	UF : 0, UT : 6,		CONFIG : 'N U T, 0, 0, 0',
	X =  -103.237  mm,	Y =   -367.062  mm,	Z =   -236.482  mm,
	W =  90.000 deg,	P =   0.000 deg,	R =   90.000 deg
};
P[2666]{
   GP1:
	UF : 0, UT : 6,		CONFIG : 'N U T, 0, 0, 0',
	X =  -103.796  mm,	Y =   -367.200  mm,	Z =   -236.035  mm,
	W =  90.000 deg,	P =   0.000 deg,	R =   90.000 deg
};
P[2667]{
   GP1:
	UF : 0, UT : 6,		CONFIG : 'N U T, 0, 0, 0',
	X =  -109.111  mm,	Y =   -370.387  mm,	Z =   -236.321  mm,
	W =  90.000 deg,	P =   0.000 deg,	R =   90.000 deg
};
P[2668]{
   GP1:
	UF : 0, UT : 6,		CONFIG : 'N U T, 0, 0, 0',
	X =  -109.874  mm,	Y =   -370.891  mm,	Z =   -236.475  mm,
	W =  90.000 deg,	P =   0.000 deg,	R =   90.000 deg
};
P[2669]{
   GP1:
	UF : 0, UT : 6,		CONFIG : 'N U T, 0, 0, 0',
	X =  -111.510  mm,	Y =   -371.847  mm,	Z =   -236.505  mm,
	W =  90.000 deg,	P =   0.000 deg,	R =   90.000 deg
};
P[2670]{
   GP1:
	UF : 0, UT : 6,		CONFIG : 'N U T, 0, 0, 0',
	X =  -113.758  mm,	Y =   -372.951  mm,	Z =   -236.032  mm,
	W =  90.000 deg,	P =   0.000 deg,	R =   90.000 deg
};
P[2671]{
   GP1:
	UF : 0, UT : 6,		CONFIG : 'N U T, 0, 0, 0',
	X =  -115.678  mm,	Y =   -374.223  mm,	Z =   -236.429  mm,
	W =  90.000 deg,	P =   0.000 deg,	R =   90.000 deg
};
P[2672]{
   GP1:
	UF : 0, UT : 6,		CONFIG : 'N U T, 0, 0, 0',
	X =  -117.192  mm,	Y =   -375.019  mm,	Z =   -236.240  mm,
	W =  90.000 deg,	P =   0.000 deg,	R =   90.000 deg
};
P[2673]{
   GP1:
	UF : 0, UT : 6,		CONFIG : 'N U T, 0, 0, 0',
	X =  -118.313  mm,	Y =   -375.755  mm,	Z =   -236.454  mm,
	W =  90.000 deg,	P =   0.000 deg,	R =   90.000 deg
};
P[2674]{
   GP1:
	UF : 0, UT : 6,		CONFIG : 'N U T, 0, 0, 0',
	X =  -120.295  mm,	Y =   -376.722  mm,	Z =   -236.025  mm,
	W =  90.000 deg,	P =   0.000 deg,	R =   90.000 deg
};
P[2675]{
   GP1:
	UF : 0, UT : 6,		CONFIG : 'N U T, 0, 0, 0',
	X =  -121.428  mm,	Y =   -377.386  mm,	Z =   -236.049  mm,
	W =  90.000 deg,	P =   0.000 deg,	R =   90.000 deg
};
P[2676]{
   GP1:
	UF : 0, UT : 6,		CONFIG : 'N U T, 0, 0, 0',
	X =  -123.033  mm,	Y =   -378.483  mm,	Z =   -236.461  mm,
	W =  90.000 deg,	P =   0.000 deg,	R =   90.000 deg
};
P[2677]{
   GP1:
	UF : 0, UT : 6,		CONFIG : 'N U T, 0, 0, 0',
	X =  -123.863  mm,	Y =   -378.861  mm,	Z =   -236.217  mm,
	W =  90.000 deg,	P =   0.000 deg,	R =   90.000 deg
};
P[2678]{
   GP1:
	UF : 0, UT : 6,		CONFIG : 'N U T, 0, 0, 0',
	X =  -125.601  mm,	Y =   -379.960  mm,	Z =   -236.448  mm,
	W =  90.000 deg,	P =   0.000 deg,	R =   90.000 deg
};
P[2679]{
   GP1:
	UF : 0, UT : 6,		CONFIG : 'N U T, 0, 0, 0',
	X =  -128.227  mm,	Y =   -381.434  mm,	Z =   -236.345  mm,
	W =  90.000 deg,	P =   0.000 deg,	R =   90.000 deg
};
P[2680]{
   GP1:
	UF : 0, UT : 6,		CONFIG : 'N U T, 0, 0, 0',
	X =  -131.933  mm,	Y =   -383.507  mm,	Z =   -236.183  mm,
	W =  90.000 deg,	P =   0.000 deg,	R =   90.000 deg
};
P[2681]{
   GP1:
	UF : 0, UT : 6,		CONFIG : 'N U T, 0, 0, 0',
	X =  -134.089  mm,	Y =   -385.044  mm,	Z =   -236.339  mm,
	W =  90.000 deg,	P =   0.000 deg,	R =   90.000 deg
};
P[2682]{
   GP1:
	UF : 0, UT : 6,		CONFIG : 'N U T, 0, 0, 0',
	X =  -136.292  mm,	Y =   -387.219  mm,	Z =   -236.419  mm,
	W =  90.000 deg,	P =   0.000 deg,	R =   90.000 deg
};
P[2683]{
   GP1:
	UF : 0, UT : 6,		CONFIG : 'N U T, 0, 0, 0',
	X =  -137.707  mm,	Y =   -389.283  mm,	Z =   -236.379  mm,
	W =  90.000 deg,	P =   0.000 deg,	R =   90.000 deg
};
P[2684]{
   GP1:
	UF : 0, UT : 6,		CONFIG : 'N U T, 0, 0, 0',
	X =  -138.543  mm,	Y =   -391.394  mm,	Z =   -236.512  mm,
	W =  90.000 deg,	P =   0.000 deg,	R =   90.000 deg
};
P[2685]{
   GP1:
	UF : 0, UT : 6,		CONFIG : 'N U T, 0, 0, 0',
	X =  -138.974  mm,	Y =   -392.288  mm,	Z =   -236.247  mm,
	W =  90.000 deg,	P =   0.000 deg,	R =   90.000 deg
};
P[2686]{
   GP1:
	UF : 0, UT : 6,		CONFIG : 'N U T, 0, 0, 0',
	X =  -139.171  mm,	Y =   -393.080  mm,	Z =   -236.154  mm,
	W =  90.000 deg,	P =   0.000 deg,	R =   90.000 deg
};
P[2687]{
   GP1:
	UF : 0, UT : 6,		CONFIG : 'N U T, 0, 0, 0',
	X =  -139.217  mm,	Y =   -394.462  mm,	Z =   -236.503  mm,
	W =  90.000 deg,	P =   0.000 deg,	R =   90.000 deg
};
P[2688]{
   GP1:
	UF : 0, UT : 6,		CONFIG : 'N U T, 0, 0, 0',
	X =  -139.347  mm,	Y =   -395.646  mm,	Z =   -236.277  mm,
	W =  90.000 deg,	P =   0.000 deg,	R =   90.000 deg
};
P[2689]{
   GP1:
	UF : 0, UT : 6,		CONFIG : 'N U T, 0, 0, 0',
	X =  -139.228  mm,	Y =   -396.334  mm,	Z =   -236.466  mm,
	W =  90.000 deg,	P =   0.000 deg,	R =   90.000 deg
};
P[2690]{
   GP1:
	UF : 0, UT : 6,		CONFIG : 'N U T, 0, 0, 0',
	X =  -139.026  mm,	Y =   -398.050  mm,	Z =   -236.504  mm,
	W =  90.000 deg,	P =   0.000 deg,	R =   90.000 deg
};
P[2691]{
   GP1:
	UF : 0, UT : 6,		CONFIG : 'N U T, 0, 0, 0',
	X =  -138.894  mm,	Y =   -399.249  mm,	Z =   -236.149  mm,
	W =  90.000 deg,	P =   0.000 deg,	R =   90.000 deg
};
P[2692]{
   GP1:
	UF : 0, UT : 6,		CONFIG : 'N U T, 0, 0, 0',
	X =  -138.534  mm,	Y =   -400.086  mm,	Z =   -236.490  mm,
	W =  90.000 deg,	P =   0.000 deg,	R =   90.000 deg
};
P[2693]{
   GP1:
	UF : 0, UT : 6,		CONFIG : 'N U T, 0, 0, 0',
	X =  -138.293  mm,	Y =   -400.993  mm,	Z =   -236.111  mm,
	W =  90.000 deg,	P =   0.000 deg,	R =   90.000 deg
};
P[2694]{
   GP1:
	UF : 0, UT : 6,		CONFIG : 'N U T, 0, 0, 0',
	X =  -132.435  mm,	Y =   -411.328  mm,	Z =   -236.323  mm,
	W =  90.000 deg,	P =   0.000 deg,	R =   90.000 deg
};
P[2695]{
   GP1:
	UF : 0, UT : 6,		CONFIG : 'N U T, 0, 0, 0',
	X =  -131.602  mm,	Y =   -412.647  mm,	Z =   -236.497  mm,
	W =  90.000 deg,	P =   0.000 deg,	R =   90.000 deg
};
P[2696]{
   GP1:
	UF : 0, UT : 6,		CONFIG : 'N U T, 0, 0, 0',
	X =  -131.076  mm,	Y =   -413.576  mm,	Z =   -236.473  mm,
	W =  90.000 deg,	P =   0.000 deg,	R =   90.000 deg
};
P[2697]{
   GP1:
	UF : 0, UT : 6,		CONFIG : 'N U T, 0, 0, 0',
	X =  -130.720  mm,	Y =   -414.277  mm,	Z =   -236.355  mm,
	W =  90.000 deg,	P =   0.000 deg,	R =   90.000 deg
};
P[2698]{
   GP1:
	UF : 0, UT : 6,		CONFIG : 'N U T, 0, 0, 0',
	X =  -129.684  mm,	Y =   -415.969  mm,	Z =   -236.496  mm,
	W =  90.000 deg,	P =   0.000 deg,	R =   90.000 deg
};
P[2699]{
   GP1:
	UF : 0, UT : 6,		CONFIG : 'N U T, 0, 0, 0',
	X =  -128.664  mm,	Y =   -417.827  mm,	Z =   -236.369  mm,
	W =  90.000 deg,	P =   0.000 deg,	R =   90.000 deg
};
P[2700]{
   GP1:
	UF : 0, UT : 6,		CONFIG : 'N U T, 0, 0, 0',
	X =  -127.347  mm,	Y =   -420.040  mm,	Z =   -236.463  mm,
	W =  90.000 deg,	P =   0.000 deg,	R =   90.000 deg
};
P[2701]{
   GP1:
	UF : 0, UT : 6,		CONFIG : 'N U T, 0, 0, 0',
	X =  -126.510  mm,	Y =   -421.475  mm,	Z =   -236.485  mm,
	W =  90.000 deg,	P =   0.000 deg,	R =   90.000 deg
};
P[2702]{
   GP1:
	UF : 0, UT : 6,		CONFIG : 'N U T, 0, 0, 0',
	X =  -125.653  mm,	Y =   -423.090  mm,	Z =   -236.300  mm,
	W =  90.000 deg,	P =   0.000 deg,	R =   90.000 deg
};
P[2703]{
   GP1:
	UF : 0, UT : 6,		CONFIG : 'N U T, 0, 0, 0',
	X =  -124.246  mm,	Y =   -425.539  mm,	Z =   -236.286  mm,
	W =  90.000 deg,	P =   0.000 deg,	R =   90.000 deg
};
P[2704]{
   GP1:
	UF : 0, UT : 6,		CONFIG : 'N U T, 0, 0, 0',
	X =  -122.328  mm,	Y =   -428.699  mm,	Z =   -236.513  mm,
	W =  90.000 deg,	P =   0.000 deg,	R =   90.000 deg
};
P[2705]{
   GP1:
	UF : 0, UT : 6,		CONFIG : 'N U T, 0, 0, 0',
	X =  -121.006  mm,	Y =   -431.158  mm,	Z =   -236.273  mm,
	W =  90.000 deg,	P =   0.000 deg,	R =   90.000 deg
};
P[2706]{
   GP1:
	UF : 0, UT : 6,		CONFIG : 'N U T, 0, 0, 0',
	X =  -117.398  mm,	Y =   -437.502  mm,	Z =   -236.140  mm,
	W =  90.000 deg,	P =   0.000 deg,	R =   90.000 deg
};
P[2707]{
   GP1:
	UF : 0, UT : 6,		CONFIG : 'N U T, 0, 0, 0',
	X =  -116.351  mm,	Y =   -439.270  mm,	Z =   -236.205  mm,
	W =  90.000 deg,	P =   0.000 deg,	R =   90.000 deg
};
P[2708]{
   GP1:
	UF : 0, UT : 6,		CONFIG : 'N U T, 0, 0, 0',
	X =  -115.892  mm,	Y =   -439.878  mm,	Z =   -236.465  mm,
	W =  90.000 deg,	P =   0.000 deg,	R =   90.000 deg
};
P[2709]{
   GP1:
	UF : 0, UT : 6,		CONFIG : 'N U T, 0, 0, 0',
	X =  -112.701  mm,	Y =   -445.426  mm,	Z =   -236.435  mm,
	W =  90.000 deg,	P =   0.000 deg,	R =   90.000 deg
};
P[2710]{
   GP1:
	UF : 0, UT : 6,		CONFIG : 'N U T, 0, 0, 0',
	X =  -111.296  mm,	Y =   -448.012  mm,	Z =   -236.222  mm,
	W =  90.000 deg,	P =   0.000 deg,	R =   90.000 deg
};
P[2711]{
   GP1:
	UF : 0, UT : 6,		CONFIG : 'N U T, 0, 0, 0',
	X =  -110.621  mm,	Y =   -448.979  mm,	Z =   -236.505  mm,
	W =  90.000 deg,	P =   0.000 deg,	R =   90.000 deg
};
P[2712]{
   GP1:
	UF : 0, UT : 6,		CONFIG : 'N U T, 0, 0, 0',
	X =  -109.896  mm,	Y =   -450.279  mm,	Z =   -236.445  mm,
	W =  90.000 deg,	P =   0.000 deg,	R =   90.000 deg
};
P[2713]{
   GP1:
	UF : 0, UT : 6,		CONFIG : 'N U T, 0, 0, 0',
	X =  -109.523  mm,	Y =   -451.116  mm,	Z =   -236.175  mm,
	W =  90.000 deg,	P =   0.000 deg,	R =   90.000 deg
};
P[2714]{
   GP1:
	UF : 0, UT : 6,		CONFIG : 'N U T, 0, 0, 0',
	X =  -109.072  mm,	Y =   -451.738  mm,	Z =   -236.398  mm,
	W =  90.000 deg,	P =   0.000 deg,	R =   90.000 deg
};
P[2715]{
   GP1:
	UF : 0, UT : 6,		CONFIG : 'N U T, 0, 0, 0',
	X =  -108.224  mm,	Y =   -453.286  mm,	Z =   -236.287  mm,
	W =  90.000 deg,	P =   0.000 deg,	R =   90.000 deg
};
P[2716]{
   GP1:
	UF : 0, UT : 6,		CONFIG : 'N U T, 0, 0, 0',
	X =  -107.392  mm,	Y =   -454.819  mm,	Z =   -236.157  mm,
	W =  90.000 deg,	P =   0.000 deg,	R =   90.000 deg
};
P[2717]{
   GP1:
	UF : 0, UT : 6,		CONFIG : 'N U T, 0, 0, 0',
	X =  -104.616  mm,	Y =   -459.487  mm,	Z =   -236.353  mm,
	W =  90.000 deg,	P =   0.000 deg,	R =   90.000 deg
};
P[2718]{
   GP1:
	UF : 0, UT : 6,		CONFIG : 'N U T, 0, 0, 0',
	X =  -103.935  mm,	Y =   -460.905  mm,	Z =   -236.019  mm,
	W =  90.000 deg,	P =   0.000 deg,	R =   90.000 deg
};
P[2719]{
   GP1:
	UF : 0, UT : 6,		CONFIG : 'N U T, 0, 0, 0',
	X =  -103.296  mm,	Y =   -461.877  mm,	Z =   -236.210  mm,
	W =  90.000 deg,	P =   0.000 deg,	R =   90.000 deg
};
P[2720]{
   GP1:
	UF : 0, UT : 6,		CONFIG : 'N U T, 0, 0, 0',
	X =  -102.498  mm,	Y =   -463.081  mm,	Z =   -236.458  mm,
	W =  90.000 deg,	P =   0.000 deg,	R =   90.000 deg
};
P[2721]{
   GP1:
	UF : 0, UT : 6,		CONFIG : 'N U T, 0, 0, 0',
	X =  -102.062  mm,	Y =   -463.796  mm,	Z =   -236.514  mm,
	W =  90.000 deg,	P =   0.000 deg,	R =   90.000 deg
};
P[2722]{
   GP1:
	UF : 0, UT : 6,		CONFIG : 'N U T, 0, 0, 0',
	X =  -98.860  mm,	Y =   -469.387  mm,	Z =   -236.452  mm,
	W =  90.000 deg,	P =   0.000 deg,	R =   90.000 deg
};
P[2723]{
   GP1:
	UF : 0, UT : 6,		CONFIG : 'N U T, 0, 0, 0',
	X =  -97.430  mm,	Y =   -472.003  mm,	Z =   -236.256  mm,
	W =  90.000 deg,	P =   0.000 deg,	R =   90.000 deg
};
P[2724]{
   GP1:
	UF : 0, UT : 6,		CONFIG : 'N U T, 0, 0, 0',
	X =  -95.657  mm,	Y =   -474.990  mm,	Z =   -236.371  mm,
	W =  90.000 deg,	P =   0.000 deg,	R =   90.000 deg
};
P[2725]{
   GP1:
	UF : 0, UT : 6,		CONFIG : 'N U T, 0, 0, 0',
	X =  -95.143  mm,	Y =   -475.820  mm,	Z =   -236.456  mm,
	W =  90.000 deg,	P =   0.000 deg,	R =   90.000 deg
};
P[2726]{
   GP1:
	UF : 0, UT : 6,		CONFIG : 'N U T, 0, 0, 0',
	X =  -94.054  mm,	Y =   -477.851  mm,	Z =   -236.254  mm,
	W =  90.000 deg,	P =   0.000 deg,	R =   90.000 deg
};
P[2727]{
   GP1:
	UF : 0, UT : 6,		CONFIG : 'N U T, 0, 0, 0',
	X =  -92.555  mm,	Y =   -480.264  mm,	Z =   -236.509  mm,
	W =  90.000 deg,	P =   0.000 deg,	R =   90.000 deg
};
P[2728]{
   GP1:
	UF : 0, UT : 6,		CONFIG : 'N U T, 0, 0, 0',
	X =  -90.494  mm,	Y =   -484.012  mm,	Z =   -236.260  mm,
	W =  90.000 deg,	P =   0.000 deg,	R =   90.000 deg
};
P[2729]{
   GP1:
	UF : 0, UT : 6,		CONFIG : 'N U T, 0, 0, 0',
	X =  -89.771  mm,	Y =   -485.179  mm,	Z =   -236.380  mm,
	W =  90.000 deg,	P =   0.000 deg,	R =   90.000 deg
};
P[2730]{
   GP1:
	UF : 0, UT : 6,		CONFIG : 'N U T, 0, 0, 0',
	X =  -88.079  mm,	Y =   -488.059  mm,	Z =   -236.451  mm,
	W =  90.000 deg,	P =   0.000 deg,	R =   90.000 deg
};
P[2731]{
   GP1:
	UF : 0, UT : 6,		CONFIG : 'N U T, 0, 0, 0',
	X =  -83.696  mm,	Y =   -495.609  mm,	Z =   -236.506  mm,
	W =  90.000 deg,	P =   0.000 deg,	R =   90.000 deg
};
P[2732]{
   GP1:
	UF : 0, UT : 6,		CONFIG : 'N U T, 0, 0, 0',
	X =  -83.326  mm,	Y =   -496.356  mm,	Z =   -236.359  mm,
	W =  90.000 deg,	P =   0.000 deg,	R =   90.000 deg
};
P[2733]{
   GP1:
	UF : 0, UT : 6,		CONFIG : 'N U T, 0, 0, 0',
	X =  -82.778  mm,	Y =   -497.396  mm,	Z =   -236.232  mm,
	W =  90.000 deg,	P =   0.000 deg,	R =   90.000 deg
};
P[2734]{
   GP1:
	UF : 0, UT : 6,		CONFIG : 'N U T, 0, 0, 0',
	X =  -82.192  mm,	Y =   -498.250  mm,	Z =   -236.458  mm,
	W =  90.000 deg,	P =   0.000 deg,	R =   90.000 deg
};
P[2735]{
   GP1:
	UF : 0, UT : 6,		CONFIG : 'N U T, 0, 0, 0',
	X =  -79.146  mm,	Y =   -503.762  mm,	Z =   -236.125  mm,
	W =  90.000 deg,	P =   0.000 deg,	R =   90.000 deg
};
P[2736]{
   GP1:
	UF : 0, UT : 6,		CONFIG : 'N U T, 0, 0, 0',
	X =  -77.301  mm,	Y =   -506.708  mm,	Z =   -236.474  mm,
	W =  90.000 deg,	P =   0.000 deg,	R =   90.000 deg
};
P[2737]{
   GP1:
	UF : 0, UT : 6,		CONFIG : 'N U T, 0, 0, 0',
	X =  -75.967  mm,	Y =   -509.301  mm,	Z =   -236.079  mm,
	W =  90.000 deg,	P =   0.000 deg,	R =   90.000 deg
};
P[2738]{
   GP1:
	UF : 0, UT : 6,		CONFIG : 'N U T, 0, 0, 0',
	X =  -74.945  mm,	Y =   -510.996  mm,	Z =   -236.183  mm,
	W =  90.000 deg,	P =   0.000 deg,	R =   90.000 deg
};
P[2739]{
   GP1:
	UF : 0, UT : 6,		CONFIG : 'N U T, 0, 0, 0',
	X =  -71.961  mm,	Y =   -516.089  mm,	Z =   -236.291  mm,
	W =  90.000 deg,	P =   0.000 deg,	R =   90.000 deg
};
P[2740]{
   GP1:
	UF : 0, UT : 6,		CONFIG : 'N U T, 0, 0, 0',
	X =  -70.926  mm,	Y =   -517.733  mm,	Z =   -236.499  mm,
	W =  90.000 deg,	P =   0.000 deg,	R =   90.000 deg
};
P[2741]{
   GP1:
	UF : 0, UT : 6,		CONFIG : 'N U T, 0, 0, 0',
	X =  -70.119  mm,	Y =   -519.466  mm,	Z =   -236.027  mm,
	W =  90.000 deg,	P =   0.000 deg,	R =   90.000 deg
};
P[2742]{
   GP1:
	UF : 0, UT : 6,		CONFIG : 'N U T, 0, 0, 0',
	X =  -67.807  mm,	Y =   -523.183  mm,	Z =   -236.430  mm,
	W =  90.000 deg,	P =   0.000 deg,	R =   90.000 deg
};
P[2743]{
   GP1:
	UF : 0, UT : 6,		CONFIG : 'N U T, 0, 0, 0',
	X =  -67.049  mm,	Y =   -524.711  mm,	Z =   -236.128  mm,
	W =  90.000 deg,	P =   0.000 deg,	R =   90.000 deg
};
P[2744]{
   GP1:
	UF : 0, UT : 6,		CONFIG : 'N U T, 0, 0, 0',
	X =  -63.701  mm,	Y =   -530.270  mm,	Z =   -236.462  mm,
	W =  90.000 deg,	P =   0.000 deg,	R =   90.000 deg
};
P[2745]{
   GP1:
	UF : 0, UT : 6,		CONFIG : 'N U T, 0, 0, 0',
	X =  -63.119  mm,	Y =   -531.321  mm,	Z =   -236.403  mm,
	W =  90.000 deg,	P =   0.000 deg,	R =   90.000 deg
};
P[2746]{
   GP1:
	UF : 0, UT : 6,		CONFIG : 'N U T, 0, 0, 0',
	X =  -61.469  mm,	Y =   -534.194  mm,	Z =   -236.385  mm,
	W =  90.000 deg,	P =   0.000 deg,	R =   90.000 deg
};
P[2747]{
   GP1:
	UF : 0, UT : 6,		CONFIG : 'N U T, 0, 0, 0',
	X =  -61.266  mm,	Y =   -534.788  mm,	Z =   -236.042  mm,
	W =  90.000 deg,	P =   0.000 deg,	R =   90.000 deg
};
P[2748]{
   GP1:
	UF : 0, UT : 6,		CONFIG : 'N U T, 0, 0, 0',
	X =  -60.082  mm,	Y =   -536.624  mm,	Z =   -236.345  mm,
	W =  90.000 deg,	P =   0.000 deg,	R =   90.000 deg
};
P[2749]{
   GP1:
	UF : 0, UT : 6,		CONFIG : 'N U T, 0, 0, 0',
	X =  -59.497  mm,	Y =   -537.677  mm,	Z =   -236.288  mm,
	W =  90.000 deg,	P =   0.000 deg,	R =   90.000 deg
};
P[2750]{
   GP1:
	UF : 0, UT : 6,		CONFIG : 'N U T, 0, 0, 0',
	X =  -59.054  mm,	Y =   -538.435  mm,	Z =   -236.301  mm,
	W =  90.000 deg,	P =   0.000 deg,	R =   90.000 deg
};
P[2751]{
   GP1:
	UF : 0, UT : 6,		CONFIG : 'N U T, 0, 0, 0',
	X =  -56.974  mm,	Y =   -542.109  mm,	Z =   -236.201  mm,
	W =  90.000 deg,	P =   0.000 deg,	R =   90.000 deg
};
P[2752]{
   GP1:
	UF : 0, UT : 6,		CONFIG : 'N U T, 0, 0, 0',
	X =  -56.447  mm,	Y =   -542.963  mm,	Z =   -236.281  mm,
	W =  90.000 deg,	P =   0.000 deg,	R =   90.000 deg
};
P[2753]{
   GP1:
	UF : 0, UT : 6,		CONFIG : 'N U T, 0, 0, 0',
	X =  -55.849  mm,	Y =   -543.939  mm,	Z =   -236.367  mm,
	W =  90.000 deg,	P =   0.000 deg,	R =   90.000 deg
};
P[2754]{
   GP1:
	UF : 0, UT : 6,		CONFIG : 'N U T, 0, 0, 0',
	X =  -54.722  mm,	Y =   -545.925  mm,	Z =   -236.316  mm,
	W =  90.000 deg,	P =   0.000 deg,	R =   90.000 deg
};
P[2755]{
   GP1:
	UF : 0, UT : 6,		CONFIG : 'N U T, 0, 0, 0',
	X =  -53.820  mm,	Y =   -547.403  mm,	Z =   -236.437  mm,
	W =  90.000 deg,	P =   0.000 deg,	R =   90.000 deg
};
P[2756]{
   GP1:
	UF : 0, UT : 6,		CONFIG : 'N U T, 0, 0, 0',
	X =  -51.903  mm,	Y =   -550.957  mm,	Z =   -236.109  mm,
	W =  90.000 deg,	P =   0.000 deg,	R =   90.000 deg
};
P[2757]{
   GP1:
	UF : 0, UT : 6,		CONFIG : 'N U T, 0, 0, 0',
	X =  -50.467  mm,	Y =   -553.413  mm,	Z =   -236.152  mm,
	W =  90.000 deg,	P =   0.000 deg,	R =   90.000 deg
};
P[2758]{
   GP1:
	UF : 0, UT : 6,		CONFIG : 'N U T, 0, 0, 0',
	X =  -49.404  mm,	Y =   -555.025  mm,	Z =   -236.475  mm,
	W =  90.000 deg,	P =   0.000 deg,	R =   90.000 deg
};
P[2759]{
   GP1:
	UF : 0, UT : 6,		CONFIG : 'N U T, 0, 0, 0',
	X =  -47.513  mm,	Y =   -558.279  mm,	Z =   -236.503  mm,
	W =  90.000 deg,	P =   0.000 deg,	R =   90.000 deg
};
P[2760]{
   GP1:
	UF : 0, UT : 6,		CONFIG : 'N U T, 0, 0, 0',
	X =  -47.011  mm,	Y =   -559.184  mm,	Z =   -236.452  mm,
	W =  90.000 deg,	P =   0.000 deg,	R =   90.000 deg
};
P[2761]{
   GP1:
	UF : 0, UT : 6,		CONFIG : 'N U T, 0, 0, 0',
	X =  -45.707  mm,	Y =   -561.524  mm,	Z =   -236.340  mm,
	W =  90.000 deg,	P =   0.000 deg,	R =   90.000 deg
};
P[2762]{
   GP1:
	UF : 0, UT : 6,		CONFIG : 'N U T, 0, 0, 0',
	X =  -44.786  mm,	Y =   -563.328  mm,	Z =   -236.045  mm,
	W =  90.000 deg,	P =   0.000 deg,	R =   90.000 deg
};
P[2763]{
   GP1:
	UF : 0, UT : 6,		CONFIG : 'N U T, 0, 0, 0',
	X =  -43.612  mm,	Y =   -565.119  mm,	Z =   -236.386  mm,
	W =  90.000 deg,	P =   0.000 deg,	R =   90.000 deg
};
P[2764]{
   GP1:
	UF : 0, UT : 6,		CONFIG : 'N U T, 0, 0, 0',
	X =  -43.076  mm,	Y =   -565.989  mm,	Z =   -236.466  mm,
	W =  90.000 deg,	P =   0.000 deg,	R =   90.000 deg
};
P[2765]{
   GP1:
	UF : 0, UT : 6,		CONFIG : 'N U T, 0, 0, 0',
	X =  -40.936  mm,	Y =   -569.844  mm,	Z =   -236.260  mm,
	W =  90.000 deg,	P =   0.000 deg,	R =   90.000 deg
};
P[2766]{
   GP1:
	UF : 0, UT : 6,		CONFIG : 'N U T, 0, 0, 0',
	X =  -40.504  mm,	Y =   -570.459  mm,	Z =   -236.446  mm,
	W =  90.000 deg,	P =   0.000 deg,	R =   90.000 deg
};
P[2767]{
   GP1:
	UF : 0, UT : 6,		CONFIG : 'N U T, 0, 0, 0',
	X =  -39.086  mm,	Y =   -572.957  mm,	Z =   -236.386  mm,
	W =  90.000 deg,	P =   0.000 deg,	R =   90.000 deg
};
P[2768]{
   GP1:
	UF : 0, UT : 6,		CONFIG : 'N U T, 0, 0, 0',
	X =  -36.165  mm,	Y =   -577.983  mm,	Z =   -236.433  mm,
	W =  90.000 deg,	P =   0.000 deg,	R =   90.000 deg
};
P[2769]{
   GP1:
	UF : 0, UT : 6,		CONFIG : 'N U T, 0, 0, 0',
	X =  -35.589  mm,	Y =   -578.926  mm,	Z =   -236.508  mm,
	W =  90.000 deg,	P =   0.000 deg,	R =   90.000 deg
};
P[2770]{
   GP1:
	UF : 0, UT : 6,		CONFIG : 'N U T, 0, 0, 0',
	X =  -30.957  mm,	Y =   -587.282  mm,	Z =   -236.040  mm,
	W =  90.000 deg,	P =   0.000 deg,	R =   90.000 deg
};
P[2771]{
   GP1:
	UF : 0, UT : 6,		CONFIG : 'N U T, 0, 0, 0',
	X =  -29.354  mm,	Y =   -589.787  mm,	Z =   -236.423  mm,
	W =  90.000 deg,	P =   0.000 deg,	R =   90.000 deg
};
P[2772]{
   GP1:
	UF : 0, UT : 6,		CONFIG : 'N U T, 0, 0, 0',
	X =  -26.877  mm,	Y =   -594.032  mm,	Z =   -236.483  mm,
	W =  90.000 deg,	P =   0.000 deg,	R =   90.000 deg
};
P[2773]{
   GP1:
	UF : 0, UT : 6,		CONFIG : 'N U T, 0, 0, 0',
	X =  -23.884  mm,	Y =   -599.221  mm,	Z =   -236.478  mm,
	W =  90.000 deg,	P =   0.000 deg,	R =   90.000 deg
};
P[2774]{
   GP1:
	UF : 0, UT : 6,		CONFIG : 'N U T, 0, 0, 0',
	X =  -22.979  mm,	Y =   -600.863  mm,	Z =   -236.375  mm,
	W =  90.000 deg,	P =   0.000 deg,	R =   90.000 deg
};
P[2775]{
   GP1:
	UF : 0, UT : 6,		CONFIG : 'N U T, 0, 0, 0',
	X =  -22.245  mm,	Y =   -602.071  mm,	Z =   -236.459  mm,
	W =  90.000 deg,	P =   0.000 deg,	R =   90.000 deg
};
P[2776]{
   GP1:
	UF : 0, UT : 6,		CONFIG : 'N U T, 0, 0, 0',
	X =  -21.779  mm,	Y =   -602.853  mm,	Z =   -236.496  mm,
	W =  90.000 deg,	P =   0.000 deg,	R =   90.000 deg
};
P[2777]{
   GP1:
	UF : 0, UT : 6,		CONFIG : 'N U T, 0, 0, 0',
	X =  -20.072  mm,	Y =   -605.860  mm,	Z =   -236.425  mm,
	W =  90.000 deg,	P =   0.000 deg,	R =   90.000 deg
};
P[2778]{
   GP1:
	UF : 0, UT : 6,		CONFIG : 'N U T, 0, 0, 0',
	X =  -17.813  mm,	Y =   -609.858  mm,	Z =   -236.308  mm,
	W =  90.000 deg,	P =   0.000 deg,	R =   90.000 deg
};
P[2779]{
   GP1:
	UF : 0, UT : 6,		CONFIG : 'N U T, 0, 0, 0',
	X =  -16.783  mm,	Y =   -611.767  mm,	Z =   -236.131  mm,
	W =  90.000 deg,	P =   0.000 deg,	R =   90.000 deg
};
P[2780]{
   GP1:
	UF : 0, UT : 6,		CONFIG : 'N U T, 0, 0, 0',
	X =  -16.133  mm,	Y =   -612.837  mm,	Z =   -236.208  mm,
	W =  90.000 deg,	P =   0.000 deg,	R =   90.000 deg
};
P[2781]{
   GP1:
	UF : 0, UT : 6,		CONFIG : 'N U T, 0, 0, 0',
	X =  -15.576  mm,	Y =   -613.717  mm,	Z =   -236.326  mm,
	W =  90.000 deg,	P =   0.000 deg,	R =   90.000 deg
};
P[2782]{
   GP1:
	UF : 0, UT : 6,		CONFIG : 'N U T, 0, 0, 0',
	X =  -13.580  mm,	Y =   -617.138  mm,	Z =   -236.378  mm,
	W =  90.000 deg,	P =   0.000 deg,	R =   90.000 deg
};
P[2783]{
   GP1:
	UF : 0, UT : 6,		CONFIG : 'N U T, 0, 0, 0',
	X =  -12.725  mm,	Y =   -618.540  mm,	Z =   -236.487  mm,
	W =  90.000 deg,	P =   0.000 deg,	R =   90.000 deg
};
P[2784]{
   GP1:
	UF : 0, UT : 6,		CONFIG : 'N U T, 0, 0, 0',
	X =  -12.420  mm,	Y =   -619.263  mm,	Z =   -236.216  mm,
	W =  90.000 deg,	P =   0.000 deg,	R =   90.000 deg
};
P[2785]{
   GP1:
	UF : 0, UT : 6,		CONFIG : 'N U T, 0, 0, 0',
	X =  -11.625  mm,	Y =   -620.474  mm,	Z =   -236.448  mm,
	W =  90.000 deg,	P =   0.000 deg,	R =   90.000 deg
};
P[2786]{
   GP1:
	UF : 0, UT : 6,		CONFIG : 'N U T, 0, 0, 0',
	X =  -8.389  mm,	Y =   -626.060  mm,	Z =   -236.474  mm,
	W =  90.000 deg,	P =   0.000 deg,	R =   90.000 deg
};
P[2787]{
   GP1:
	UF : 0, UT : 6,		CONFIG : 'N U T, 0, 0, 0',
	X =  -6.891  mm,	Y =   -628.784  mm,	Z =   -236.289  mm,
	W =  90.000 deg,	P =   0.000 deg,	R =   90.000 deg
};
P[2788]{
   GP1:
	UF : 0, UT : 6,		CONFIG : 'N U T, 0, 0, 0',
	X =  -6.304  mm,	Y =   -629.768  mm,	Z =   -236.336  mm,
	W =  90.000 deg,	P =   0.000 deg,	R =   90.000 deg
};
P[2789]{
   GP1:
	UF : 0, UT : 6,		CONFIG : 'N U T, 0, 0, 0',
	X =  -5.756  mm,	Y =   -630.621  mm,	Z =   -236.473  mm,
	W =  90.000 deg,	P =   0.000 deg,	R =   90.000 deg
};
P[2790]{
   GP1:
	UF : 0, UT : 6,		CONFIG : 'N U T, 0, 0, 0',
	X =  -3.081  mm,	Y =   -635.232  mm,	Z =   -236.502  mm,
	W =  90.000 deg,	P =   0.000 deg,	R =   90.000 deg
};
P[2791]{
   GP1:
	UF : 0, UT : 6,		CONFIG : 'N U T, 0, 0, 0',
	X =  -2.279  mm,	Y =   -636.663  mm,	Z =   -236.443  mm,
	W =  90.000 deg,	P =   0.000 deg,	R =   90.000 deg
};
P[2792]{
   GP1:
	UF : 0, UT : 6,		CONFIG : 'N U T, 0, 0, 0',
	X =  -0.761  mm,	Y =   -639.336  mm,	Z =   -236.383  mm,
	W =  90.000 deg,	P =   0.000 deg,	R =   90.000 deg
};
P[2793]{
   GP1:
	UF : 0, UT : 6,		CONFIG : 'N U T, 0, 0, 0',
	X =  0.858  mm,	Y =   -642.148  mm,	Z =   -236.369  mm,
	W =  90.000 deg,	P =   0.000 deg,	R =   90.000 deg
};
P[2794]{
   GP1:
	UF : 0, UT : 6,		CONFIG : 'N U T, 0, 0, 0',
	X =  1.759  mm,	Y =   -643.769  mm,	Z =   -236.287  mm,
	W =  90.000 deg,	P =   0.000 deg,	R =   90.000 deg
};
P[2795]{
   GP1:
	UF : 0, UT : 6,		CONFIG : 'N U T, 0, 0, 0',
	X =  3.576  mm,	Y =   -646.947  mm,	Z =   -236.243  mm,
	W =  90.000 deg,	P =   0.000 deg,	R =   90.000 deg
};
P[2796]{
   GP1:
	UF : 0, UT : 6,		CONFIG : 'N U T, 0, 0, 0',
	X =  4.161  mm,	Y =   -647.944  mm,	Z =   -236.266  mm,
	W =  90.000 deg,	P =   0.000 deg,	R =   90.000 deg
};
P[2797]{
   GP1:
	UF : 0, UT : 6,		CONFIG : 'N U T, 0, 0, 0',
	X =  4.658  mm,	Y =   -648.779  mm,	Z =   -236.302  mm,
	W =  90.000 deg,	P =   0.000 deg,	R =   90.000 deg
};
P[2798]{
   GP1:
	UF : 0, UT : 6,		CONFIG : 'N U T, 0, 0, 0',
	X =  5.200  mm,	Y =   -649.689  mm,	Z =   -236.343  mm,
	W =  90.000 deg,	P =   0.000 deg,	R =   90.000 deg
};
P[2799]{
   GP1:
	UF : 0, UT : 6,		CONFIG : 'N U T, 0, 0, 0',
	X =  5.838  mm,	Y =   -650.769  mm,	Z =   -236.379  mm,
	W =  90.000 deg,	P =   0.000 deg,	R =   90.000 deg
};
P[2800]{
   GP1:
	UF : 0, UT : 6,		CONFIG : 'N U T, 0, 0, 0',
	X =  9.409  mm,	Y =   -656.940  mm,	Z =   -236.398  mm,
	W =  90.000 deg,	P =   0.000 deg,	R =   90.000 deg
};
P[2801]{
   GP1:
	UF : 0, UT : 6,		CONFIG : 'N U T, 0, 0, 0',
	X =  11.270  mm,	Y =   -660.160  mm,	Z =   -236.402  mm,
	W =  90.000 deg,	P =   0.000 deg,	R =   90.000 deg
};
P[2802]{
   GP1:
	UF : 0, UT : 6,		CONFIG : 'N U T, 0, 0, 0',
	X =  12.634  mm,	Y =   -662.517  mm,	Z =   -236.408  mm,
	W =  90.000 deg,	P =   0.000 deg,	R =   90.000 deg
};
P[2803]{
   GP1:
	UF : 0, UT : 6,		CONFIG : 'N U T, 0, 0, 0',
	X =  13.698  mm,	Y =   -664.325  mm,	Z =   -236.457  mm,
	W =  90.000 deg,	P =   0.000 deg,	R =   90.000 deg
};
P[2804]{
   GP1:
	UF : 0, UT : 6,		CONFIG : 'N U T, 0, 0, 0',
	X =  14.024  mm,	Y =   -665.020  mm,	Z =   -236.275  mm,
	W =  90.000 deg,	P =   0.000 deg,	R =   90.000 deg
};
P[2805]{
   GP1:
	UF : 0, UT : 6,		CONFIG : 'N U T, 0, 0, 0',
	X =  15.603  mm,	Y =   -667.779  mm,	Z =   -236.241  mm,
	W =  90.000 deg,	P =   0.000 deg,	R =   90.000 deg
};
P[2806]{
   GP1:
	UF : 0, UT : 6,		CONFIG : 'N U T, 0, 0, 0',
	X =  16.111  mm,	Y =   -668.721  mm,	Z =   -236.153  mm,
	W =  90.000 deg,	P =   0.000 deg,	R =   90.000 deg
};
P[2807]{
   GP1:
	UF : 0, UT : 6,		CONFIG : 'N U T, 0, 0, 0',
	X =  16.623  mm,	Y =   -669.667  mm,	Z =   -236.072  mm,
	W =  90.000 deg,	P =   0.000 deg,	R =   90.000 deg
};
P[2808]{
   GP1:
	UF : 0, UT : 6,		CONFIG : 'N U T, 0, 0, 0',
	X =  18.028  mm,	Y =   -672.101  mm,	Z =   -236.068  mm,
	W =  90.000 deg,	P =   0.000 deg,	R =   90.000 deg
};
P[2809]{
   GP1:
	UF : 0, UT : 6,		CONFIG : 'N U T, 0, 0, 0',
	X =  18.530  mm,	Y =   -672.742  mm,	Z =   -236.391  mm,
	W =  90.000 deg,	P =   0.000 deg,	R =   90.000 deg
};
P[2810]{
   GP1:
	UF : 0, UT : 6,		CONFIG : 'N U T, 0, 0, 0',
	X =  20.590  mm,	Y =   -676.325  mm,	Z =   -236.365  mm,
	W =  90.000 deg,	P =   0.000 deg,	R =   90.000 deg
};
P[2811]{
   GP1:
	UF : 0, UT : 6,		CONFIG : 'N U T, 0, 0, 0',
	X =  22.083  mm,	Y =   -679.038  mm,	Z =   -236.189  mm,
	W =  90.000 deg,	P =   0.000 deg,	R =   90.000 deg
};
P[2812]{
   GP1:
	UF : 0, UT : 6,		CONFIG : 'N U T, 0, 0, 0',
	X =  23.478  mm,	Y =   -681.252  mm,	Z =   -236.473  mm,
	W =  90.000 deg,	P =   0.000 deg,	R =   90.000 deg
};
P[2813]{
   GP1:
	UF : 0, UT : 6,		CONFIG : 'N U T, 0, 0, 0',
	X =  24.055  mm,	Y =   -682.577  mm,	Z =   -236.016  mm,
	W =  90.000 deg,	P =   0.000 deg,	R =   90.000 deg
};
P[2814]{
   GP1:
	UF : 0, UT : 6,		CONFIG : 'N U T, 0, 0, 0',
	X =  27.203  mm,	Y =   -687.875  mm,	Z =   -236.234  mm,
	W =  90.000 deg,	P =   0.000 deg,	R =   90.000 deg
};
P[2815]{
   GP1:
	UF : 0, UT : 6,		CONFIG : 'N U T, 0, 0, 0',
	X =  27.873  mm,	Y =   -688.847  mm,	Z =   -236.496  mm,
	W =  90.000 deg,	P =   0.000 deg,	R =   90.000 deg
};
P[2816]{
   GP1:
	UF : 0, UT : 6,		CONFIG : 'N U T, 0, 0, 0',
	X =  28.459  mm,	Y =   -689.879  mm,	Z =   -236.471  mm,
	W =  90.000 deg,	P =   0.000 deg,	R =   90.000 deg
};
P[2817]{
   GP1:
	UF : 0, UT : 6,		CONFIG : 'N U T, 0, 0, 0',
	X =  29.323  mm,	Y =   -691.489  mm,	Z =   -236.312  mm,
	W =  90.000 deg,	P =   0.000 deg,	R =   90.000 deg
};
P[2818]{
   GP1:
	UF : 0, UT : 6,		CONFIG : 'N U T, 0, 0, 0',
	X =  30.796  mm,	Y =   -694.114  mm,	Z =   -236.209  mm,
	W =  90.000 deg,	P =   0.000 deg,	R =   90.000 deg
};
P[2819]{
   GP1:
	UF : 0, UT : 6,		CONFIG : 'N U T, 0, 0, 0',
	X =  32.101  mm,	Y =   -696.258  mm,	Z =   -236.372  mm,
	W =  90.000 deg,	P =   0.000 deg,	R =   90.000 deg
};
P[2820]{
   GP1:
	UF : 0, UT : 6,		CONFIG : 'N U T, 0, 0, 0',
	X =  34.273  mm,	Y =   -699.958  mm,	Z =   -236.458  mm,
	W =  90.000 deg,	P =   0.000 deg,	R =   90.000 deg
};
P[2821]{
   GP1:
	UF : 0, UT : 6,		CONFIG : 'N U T, 0, 0, 0',
	X =  35.034  mm,	Y =   -701.310  mm,	Z =   -236.409  mm,
	W =  90.000 deg,	P =   0.000 deg,	R =   90.000 deg
};
P[2822]{
   GP1:
	UF : 0, UT : 6,		CONFIG : 'N U T, 0, 0, 0',
	X =  35.645  mm,	Y =   -702.304  mm,	Z =   -236.268  mm,
	W =  90.000 deg,	P =   0.000 deg,	R =   90.000 deg
};
P[2823]{
   GP1:
	UF : 0, UT : 6,		CONFIG : 'N U T, 0, 0, 0',
	X =  36.316  mm,	Y =   -703.207  mm,	Z =   -236.328  mm,
	W =  90.000 deg,	P =   0.000 deg,	R =   90.000 deg
};
P[2824]{
   GP1:
	UF : 0, UT : 6,		CONFIG : 'N U T, 0, 0, 0',
	X =  37.230  mm,	Y =   -704.410  mm,	Z =   -236.133  mm,
	W =  90.000 deg,	P =   0.000 deg,	R =   90.000 deg
};
P[2825]{
   GP1:
	UF : 0, UT : 6,		CONFIG : 'N U T, 0, 0, 0',
	X =  38.416  mm,	Y =   -705.323  mm,	Z =   -236.491  mm,
	W =  90.000 deg,	P =   0.000 deg,	R =   90.000 deg
};
P[2826]{
   GP1:
	UF : 0, UT : 6,		CONFIG : 'N U T, 0, 0, 0',
	X =  39.372  mm,	Y =   -706.033  mm,	Z =   -236.512  mm,
	W =  90.000 deg,	P =   0.000 deg,	R =   90.000 deg
};
P[2827]{
   GP1:
	UF : 0, UT : 6,		CONFIG : 'N U T, 0, 0, 0',
	X =  40.316  mm,	Y =   -706.802  mm,	Z =   -236.215  mm,
	W =  90.000 deg,	P =   0.000 deg,	R =   90.000 deg
};
P[2828]{
   GP1:
	UF : 0, UT : 6,		CONFIG : 'N U T, 0, 0, 0',
	X =  45.468  mm,	Y =   -708.560  mm,	Z =   -236.089  mm,
	W =  90.000 deg,	P =   0.000 deg,	R =   90.000 deg
};
P[2829]{
   GP1:
	UF : 0, UT : 6,		CONFIG : 'N U T, 0, 0, 0',
	X =  46.166  mm,	Y =   -708.584  mm,	Z =   -236.188  mm,
	W =  90.000 deg,	P =   0.000 deg,	R =   90.000 deg
};
P[2830]{
   GP1:
	UF : 0, UT : 6,		CONFIG : 'N U T, 0, 0, 0',
	X =  47.620  mm,	Y =   -708.412  mm,	Z =   -236.473  mm,
	W =  90.000 deg,	P =   0.000 deg,	R =   90.000 deg
};
P[2831]{
   GP1:
	UF : 0, UT : 6,		CONFIG : 'N U T, 0, 0, 0',
	X =  48.514  mm,	Y =   -708.561  mm,	Z =   -236.085  mm,
	W =  90.000 deg,	P =   0.000 deg,	R =   90.000 deg
};
P[2832]{
   GP1:
	UF : 0, UT : 6,		CONFIG : 'N U T, 0, 0, 0',
	X =  49.691  mm,	Y =   -708.218  mm,	Z =   -236.321  mm,
	W =  90.000 deg,	P =   0.000 deg,	R =   90.000 deg
};
P[2833]{
   GP1:
	UF : 0, UT : 6,		CONFIG : 'N U T, 0, 0, 0',
	X =  52.176  mm,	Y =   -707.394  mm,	Z =   -236.458  mm,
	W =  90.000 deg,	P =   0.000 deg,	R =   90.000 deg
};
P[2834]{
   GP1:
	UF : 0, UT : 6,		CONFIG : 'N U T, 0, 0, 0',
	X =  56.284  mm,	Y =   -705.282  mm,	Z =   -236.360  mm,
	W =  90.000 deg,	P =   0.000 deg,	R =   90.000 deg
};
P[2835]{
   GP1:
	UF : 0, UT : 6,		CONFIG : 'N U T, 0, 0, 0',
	X =  59.075  mm,	Y =   -703.766  mm,	Z =   -236.129  mm,
	W =  90.000 deg,	P =   0.000 deg,	R =   90.000 deg
};
P[2836]{
   GP1:
	UF : 0, UT : 6,		CONFIG : 'N U T, 0, 0, 0',
	X =  59.898  mm,	Y =   -703.189  mm,	Z =   -236.376  mm,
	W =  90.000 deg,	P =   0.000 deg,	R =   90.000 deg
};
P[2837]{
   GP1:
	UF : 0, UT : 6,		CONFIG : 'N U T, 0, 0, 0',
	X =  61.634  mm,	Y =   -702.160  mm,	Z =   -236.438  mm,
	W =  90.000 deg,	P =   0.000 deg,	R =   90.000 deg
};
P[2838]{
   GP1:
	UF : 0, UT : 6,		CONFIG : 'N U T, 0, 0, 0',
	X =  63.182  mm,	Y =   -701.329  mm,	Z =   -236.288  mm,
	W =  90.000 deg,	P =   0.000 deg,	R =   90.000 deg
};
P[2839]{
   GP1:
	UF : 0, UT : 6,		CONFIG : 'N U T, 0, 0, 0',
	X =  66.400  mm,	Y =   -699.411  mm,	Z =   -236.431  mm,
	W =  90.000 deg,	P =   0.000 deg,	R =   90.000 deg
};
P[2840]{
   GP1:
	UF : 0, UT : 6,		CONFIG : 'N U T, 0, 0, 0',
	X =  68.844  mm,	Y =   -698.171  mm,	Z =   -236.017  mm,
	W =  90.000 deg,	P =   0.000 deg,	R =   90.000 deg
};
P[2841]{
   GP1:
	UF : 0, UT : 6,		CONFIG : 'N U T, 0, 0, 0',
	X =  69.752  mm,	Y =   -697.447  mm,	Z =   -236.500  mm,
	W =  90.000 deg,	P =   0.000 deg,	R =   90.000 deg
};
P[2842]{
   GP1:
	UF : 0, UT : 6,		CONFIG : 'N U T, 0, 0, 0',
	X =  71.033  mm,	Y =   -696.871  mm,	Z =   -236.105  mm,
	W =  90.000 deg,	P =   0.000 deg,	R =   90.000 deg
};
P[2843]{
   GP1:
	UF : 0, UT : 6,		CONFIG : 'N U T, 0, 0, 0',
	X =  79.303  mm,	Y =   -692.067  mm,	Z =   -236.174  mm,
	W =  90.000 deg,	P =   0.000 deg,	R =   90.000 deg
};
P[2844]{
   GP1:
	UF : 0, UT : 6,		CONFIG : 'N U T, 0, 0, 0',
	X =  80.219  mm,	Y =   -691.581  mm,	Z =   -236.072  mm,
	W =  90.000 deg,	P =   0.000 deg,	R =   90.000 deg
};
P[2845]{
   GP1:
	UF : 0, UT : 6,		CONFIG : 'N U T, 0, 0, 0',
	X =  82.107  mm,	Y =   -690.492  mm,	Z =   -236.067  mm,
	W =  90.000 deg,	P =   0.000 deg,	R =   90.000 deg
};
P[2846]{
   GP1:
	UF : 0, UT : 6,		CONFIG : 'N U T, 0, 0, 0',
	X =  82.790  mm,	Y =   -689.951  mm,	Z =   -236.423  mm,
	W =  90.000 deg,	P =   0.000 deg,	R =   90.000 deg
};
P[2847]{
   GP1:
	UF : 0, UT : 6,		CONFIG : 'N U T, 0, 0, 0',
	X =  84.311  mm,	Y =   -689.078  mm,	Z =   -236.410  mm,
	W =  90.000 deg,	P =   0.000 deg,	R =   90.000 deg
};
P[2848]{
   GP1:
	UF : 0, UT : 6,		CONFIG : 'N U T, 0, 0, 0',
	X =  87.841  mm,	Y =   -687.160  mm,	Z =   -236.120  mm,
	W =  90.000 deg,	P =   0.000 deg,	R =   90.000 deg
};
P[2849]{
   GP1:
	UF : 0, UT : 6,		CONFIG : 'N U T, 0, 0, 0',
	X =  90.417  mm,	Y =   -685.662  mm,	Z =   -236.144  mm,
	W =  90.000 deg,	P =   0.000 deg,	R =   90.000 deg
};
P[2850]{
   GP1:
	UF : 0, UT : 6,		CONFIG : 'N U T, 0, 0, 0',
	X =  92.018  mm,	Y =   -684.683  mm,	Z =   -236.277  mm,
	W =  90.000 deg,	P =   0.000 deg,	R =   90.000 deg
};
P[2851]{
   GP1:
	UF : 0, UT : 6,		CONFIG : 'N U T, 0, 0, 0',
	X =  95.149  mm,	Y =   -682.789  mm,	Z =   -236.487  mm,
	W =  90.000 deg,	P =   0.000 deg,	R =   90.000 deg
};
P[2852]{
   GP1:
	UF : 0, UT : 6,		CONFIG : 'N U T, 0, 0, 0',
	X =  96.225  mm,	Y =   -682.338  mm,	Z =   -236.074  mm,
	W =  90.000 deg,	P =   0.000 deg,	R =   90.000 deg
};
P[2853]{
   GP1:
	UF : 0, UT : 6,		CONFIG : 'N U T, 0, 0, 0',
	X =  97.254  mm,	Y =   -681.639  mm,	Z =   -236.329  mm,
	W =  90.000 deg,	P =   0.000 deg,	R =   90.000 deg
};
P[2854]{
   GP1:
	UF : 0, UT : 6,		CONFIG : 'N U T, 0, 0, 0',
	X =  97.958  mm,	Y =   -681.341  mm,	Z =   -236.066  mm,
	W =  90.000 deg,	P =   0.000 deg,	R =   90.000 deg
};
P[2855]{
   GP1:
	UF : 0, UT : 6,		CONFIG : 'N U T, 0, 0, 0',
	X =  109.694  mm,	Y =   -674.564  mm,	Z =   -236.067  mm,
	W =  90.000 deg,	P =   0.000 deg,	R =   90.000 deg
};
P[2856]{
   GP1:
	UF : 0, UT : 6,		CONFIG : 'N U T, 0, 0, 0',
	X =  114.432  mm,	Y =   -671.794  mm,	Z =   -236.150  mm,
	W =  90.000 deg,	P =   0.000 deg,	R =   90.000 deg
};
P[2857]{
   GP1:
	UF : 0, UT : 6,		CONFIG : 'N U T, 0, 0, 0',
	X =  118.155  mm,	Y =   -669.576  mm,	Z =   -236.314  mm,
	W =  90.000 deg,	P =   0.000 deg,	R =   90.000 deg
};
P[2858]{
   GP1:
	UF : 0, UT : 6,		CONFIG : 'N U T, 0, 0, 0',
	X =  119.202  mm,	Y =   -668.923  mm,	Z =   -236.432  mm,
	W =  90.000 deg,	P =   0.000 deg,	R =   90.000 deg
};
P[2859]{
   GP1:
	UF : 0, UT : 6,		CONFIG : 'N U T, 0, 0, 0',
	X =  124.199  mm,	Y =   -666.158  mm,	Z =   -236.141  mm,
	W =  90.000 deg,	P =   0.000 deg,	R =   90.000 deg
};
P[2860]{
   GP1:
	UF : 0, UT : 6,		CONFIG : 'N U T, 0, 0, 0',
	X =  128.547  mm,	Y =   -663.511  mm,	Z =   -236.473  mm,
	W =  90.000 deg,	P =   0.000 deg,	R =   90.000 deg
};
P[2861]{
   GP1:
	UF : 0, UT : 6,		CONFIG : 'N U T, 0, 0, 0',
	X =  130.385  mm,	Y =   -662.451  mm,	Z =   -236.470  mm,
	W =  90.000 deg,	P =   0.000 deg,	R =   90.000 deg
};
P[2862]{
   GP1:
	UF : 0, UT : 6,		CONFIG : 'N U T, 0, 0, 0',
	X =  131.198  mm,	Y =   -662.021  mm,	Z =   -236.374  mm,
	W =  90.000 deg,	P =   0.000 deg,	R =   90.000 deg
};
P[2863]{
   GP1:
	UF : 0, UT : 6,		CONFIG : 'N U T, 0, 0, 0',
	X =  133.444  mm,	Y =   -660.671  mm,	Z =   -236.505  mm,
	W =  90.000 deg,	P =   0.000 deg,	R =   90.000 deg
};
P[2864]{
   GP1:
	UF : 0, UT : 6,		CONFIG : 'N U T, 0, 0, 0',
	X =  136.895  mm,	Y =   -658.782  mm,	Z =   -236.252  mm,
	W =  90.000 deg,	P =   0.000 deg,	R =   90.000 deg
};
P[2865]{
   GP1:
	UF : 0, UT : 6,		CONFIG : 'N U T, 0, 0, 0',
	X =  139.530  mm,	Y =   -657.201  mm,	Z =   -236.398  mm,
	W =  90.000 deg,	P =   0.000 deg,	R =   90.000 deg
};
P[2866]{
   GP1:
	UF : 0, UT : 6,		CONFIG : 'N U T, 0, 0, 0',
	X =  140.472  mm,	Y =   -656.701  mm,	Z =   -236.291  mm,
	W =  90.000 deg,	P =   0.000 deg,	R =   90.000 deg
};
P[2867]{
   GP1:
	UF : 0, UT : 6,		CONFIG : 'N U T, 0, 0, 0',
	X =  142.309  mm,	Y =   -655.675  mm,	Z =   -236.206  mm,
	W =  90.000 deg,	P =   0.000 deg,	R =   90.000 deg
};
P[2868]{
   GP1:
	UF : 0, UT : 6,		CONFIG : 'N U T, 0, 0, 0',
	X =  144.452  mm,	Y =   -654.460  mm,	Z =   -236.153  mm,
	W =  90.000 deg,	P =   0.000 deg,	R =   90.000 deg
};
P[2869]{
   GP1:
	UF : 0, UT : 6,		CONFIG : 'N U T, 0, 0, 0',
	X =  145.368  mm,	Y =   -653.865  mm,	Z =   -236.312  mm,
	W =  90.000 deg,	P =   0.000 deg,	R =   90.000 deg
};
P[2870]{
   GP1:
	UF : 0, UT : 6,		CONFIG : 'N U T, 0, 0, 0',
	X =  148.587  mm,	Y =   -652.078  mm,	Z =   -236.139  mm,
	W =  90.000 deg,	P =   0.000 deg,	R =   90.000 deg
};
P[2871]{
   GP1:
	UF : 0, UT : 6,		CONFIG : 'N U T, 0, 0, 0',
	X =  150.438  mm,	Y =   -650.983  mm,	Z =   -236.201  mm,
	W =  90.000 deg,	P =   0.000 deg,	R =   90.000 deg
};
P[2872]{
   GP1:
	UF : 0, UT : 6,		CONFIG : 'N U T, 0, 0, 0',
	X =  152.235  mm,	Y =   -649.851  mm,	Z =   -236.430  mm,
	W =  90.000 deg,	P =   0.000 deg,	R =   90.000 deg
};
P[2873]{
   GP1:
	UF : 0, UT : 6,		CONFIG : 'N U T, 0, 0, 0',
	X =  154.556  mm,	Y =   -648.513  mm,	Z =   -236.428  mm,
	W =  90.000 deg,	P =   0.000 deg,	R =   90.000 deg
};
P[2874]{
   GP1:
	UF : 0, UT : 6,		CONFIG : 'N U T, 0, 0, 0',
	X =  155.199  mm,	Y =   -648.213  mm,	Z =   -236.255  mm,
	W =  90.000 deg,	P =   0.000 deg,	R =   90.000 deg
};
P[2875]{
   GP1:
	UF : 0, UT : 6,		CONFIG : 'N U T, 0, 0, 0',
	X =  157.457  mm,	Y =   -646.981  mm,	Z =   -236.079  mm,
	W =  90.000 deg,	P =   0.000 deg,	R =   90.000 deg
};
P[2876]{
   GP1:
	UF : 0, UT : 6,		CONFIG : 'N U T, 0, 0, 0',
	X =  159.587  mm,	Y =   -645.594  mm,	Z =   -236.459  mm,
	W =  90.000 deg,	P =   0.000 deg,	R =   90.000 deg
};
P[2877]{
   GP1:
	UF : 0, UT : 6,		CONFIG : 'N U T, 0, 0, 0',
	X =  160.338  mm,	Y =   -645.329  mm,	Z =   -236.051  mm,
	W =  90.000 deg,	P =   0.000 deg,	R =   90.000 deg
};
P[2878]{
   GP1:
	UF : 0, UT : 6,		CONFIG : 'N U T, 0, 0, 0',
	X =  163.247  mm,	Y =   -643.545  mm,	Z =   -236.305  mm,
	W =  90.000 deg,	P =   0.000 deg,	R =   90.000 deg
};
P[2879]{
   GP1:
	UF : 0, UT : 6,		CONFIG : 'N U T, 0, 0, 0',
	X =  163.919  mm,	Y =   -643.248  mm,	Z =   -236.085  mm,
	W =  90.000 deg,	P =   0.000 deg,	R =   90.000 deg
};
P[2880]{
   GP1:
	UF : 0, UT : 6,		CONFIG : 'N U T, 0, 0, 0',
	X =  165.705  mm,	Y =   -642.087  mm,	Z =   -236.398  mm,
	W =  90.000 deg,	P =   0.000 deg,	R =   90.000 deg
};
P[2881]{
   GP1:
	UF : 0, UT : 6,		CONFIG : 'N U T, 0, 0, 0',
	X =  167.372  mm,	Y =   -641.217  mm,	Z =   -236.176  mm,
	W =  90.000 deg,	P =   0.000 deg,	R =   90.000 deg
};
P[2882]{
   GP1:
	UF : 0, UT : 6,		CONFIG : 'N U T, 0, 0, 0',
	X =  168.552  mm,	Y =   -640.521  mm,	Z =   -236.212  mm,
	W =  90.000 deg,	P =   0.000 deg,	R =   90.000 deg
};
P[2883]{
   GP1:
	UF : 0, UT : 6,		CONFIG : 'N U T, 0, 0, 0',
	X =  169.884  mm,	Y =   -639.665  mm,	Z =   -236.422  mm,
	W =  90.000 deg,	P =   0.000 deg,	R =   90.000 deg
};
P[2884]{
   GP1:
	UF : 0, UT : 6,		CONFIG : 'N U T, 0, 0, 0',
	X =  171.046  mm,	Y =   -639.027  mm,	Z =   -236.340  mm,
	W =  90.000 deg,	P =   0.000 deg,	R =   90.000 deg
};
P[2885]{
   GP1:
	UF : 0, UT : 6,		CONFIG : 'N U T, 0, 0, 0',
	X =  173.896  mm,	Y =   -637.386  mm,	Z =   -236.330  mm,
	W =  90.000 deg,	P =   0.000 deg,	R =   90.000 deg
};
P[2886]{
   GP1:
	UF : 0, UT : 6,		CONFIG : 'N U T, 0, 0, 0',
	X =  175.734  mm,	Y =   -636.399  mm,	Z =   -236.152  mm,
	W =  90.000 deg,	P =   0.000 deg,	R =   90.000 deg
};
P[2887]{
   GP1:
	UF : 0, UT : 6,		CONFIG : 'N U T, 0, 0, 0',
	X =  178.103  mm,	Y =   -634.901  mm,	Z =   -236.465  mm,
	W =  90.000 deg,	P =   0.000 deg,	R =   90.000 deg
};
P[2888]{
   GP1:
	UF : 0, UT : 6,		CONFIG : 'N U T, 0, 0, 0',
	X =  179.069  mm,	Y =   -634.471  mm,	Z =   -236.155  mm,
	W =  90.000 deg,	P =   0.000 deg,	R =   90.000 deg
};
P[2889]{
   GP1:
	UF : 0, UT : 6,		CONFIG : 'N U T, 0, 0, 0',
	X =  180.259  mm,	Y =   -633.839  mm,	Z =   -236.021  mm,
	W =  90.000 deg,	P =   0.000 deg,	R =   90.000 deg
};
P[2890]{
   GP1:
	UF : 0, UT : 6,		CONFIG : 'N U T, 0, 0, 0',
	X =  181.350  mm,	Y =   -633.209  mm,	Z =   -236.022  mm,
	W =  90.000 deg,	P =   0.000 deg,	R =   90.000 deg
};
P[2891]{
   GP1:
	UF : 0, UT : 6,		CONFIG : 'N U T, 0, 0, 0',
	X =  188.115  mm,	Y =   -629.190  mm,	Z =   -236.296  mm,
	W =  90.000 deg,	P =   0.000 deg,	R =   90.000 deg
};
P[2892]{
   GP1:
	UF : 0, UT : 6,		CONFIG : 'N U T, 0, 0, 0',
	X =  194.718  mm,	Y =   -625.303  mm,	Z =   -236.477  mm,
	W =  90.000 deg,	P =   0.000 deg,	R =   90.000 deg
};
P[2893]{
   GP1:
	UF : 0, UT : 6,		CONFIG : 'N U T, 0, 0, 0',
	X =  195.641  mm,	Y =   -624.763  mm,	Z =   -236.494  mm,
	W =  90.000 deg,	P =   0.000 deg,	R =   90.000 deg
};
P[2894]{
   GP1:
	UF : 0, UT : 6,		CONFIG : 'N U T, 0, 0, 0',
	X =  196.542  mm,	Y =   -624.285  mm,	Z =   -236.391  mm,
	W =  90.000 deg,	P =   0.000 deg,	R =   90.000 deg
};
P[2895]{
   GP1:
	UF : 0, UT : 6,		CONFIG : 'N U T, 0, 0, 0',
	X =  198.006  mm,	Y =   -623.439  mm,	Z =   -236.393  mm,
	W =  90.000 deg,	P =   0.000 deg,	R =   90.000 deg
};
P[2896]{
   GP1:
	UF : 0, UT : 6,		CONFIG : 'N U T, 0, 0, 0',
	X =  198.990  mm,	Y =   -622.855  mm,	Z =   -236.432  mm,
	W =  90.000 deg,	P =   0.000 deg,	R =   90.000 deg
};
P[2897]{
   GP1:
	UF : 0, UT : 6,		CONFIG : 'N U T, 0, 0, 0',
	X =  201.991  mm,	Y =   -621.238  mm,	Z =   -236.150  mm,
	W =  90.000 deg,	P =   0.000 deg,	R =   90.000 deg
};
P[2898]{
   GP1:
	UF : 0, UT : 6,		CONFIG : 'N U T, 0, 0, 0',
	X =  203.362  mm,	Y =   -620.476  mm,	Z =   -236.080  mm,
	W =  90.000 deg,	P =   0.000 deg,	R =   90.000 deg
};
P[2899]{
   GP1:
	UF : 0, UT : 6,		CONFIG : 'N U T, 0, 0, 0',
	X =  205.942  mm,	Y =   -618.867  mm,	Z =   -236.366  mm,
	W =  90.000 deg,	P =   0.000 deg,	R =   90.000 deg
};
P[2900]{
   GP1:
	UF : 0, UT : 6,		CONFIG : 'N U T, 0, 0, 0',
	X =  206.618  mm,	Y =   -618.506  mm,	Z =   -236.298  mm,
	W =  90.000 deg,	P =   0.000 deg,	R =   90.000 deg
};
P[2901]{
   GP1:
	UF : 0, UT : 6,		CONFIG : 'N U T, 0, 0, 0',
	X =  208.093  mm,	Y =   -617.590  mm,	Z =   -236.453  mm,
	W =  90.000 deg,	P =   0.000 deg,	R =   90.000 deg
};
P[2902]{
   GP1:
	UF : 0, UT : 6,		CONFIG : 'N U T, 0, 0, 0',
	X =  209.850  mm,	Y =   -616.555  mm,	Z =   -236.502  mm,
	W =  90.000 deg,	P =   0.000 deg,	R =   90.000 deg
};
P[2903]{
   GP1:
	UF : 0, UT : 6,		CONFIG : 'N U T, 0, 0, 0',
	X =  211.605  mm,	Y =   -615.684  mm,	Z =   -236.157  mm,
	W =  90.000 deg,	P =   0.000 deg,	R =   90.000 deg
};
P[2904]{
   GP1:
	UF : 0, UT : 6,		CONFIG : 'N U T, 0, 0, 0',
	X =  212.954  mm,	Y =   -614.933  mm,	Z =   -236.090  mm,
	W =  90.000 deg,	P =   0.000 deg,	R =   90.000 deg
};
P[2905]{
   GP1:
	UF : 0, UT : 6,		CONFIG : 'N U T, 0, 0, 0',
	X =  214.059  mm,	Y =   -614.147  mm,	Z =   -236.449  mm,
	W =  90.000 deg,	P =   0.000 deg,	R =   90.000 deg
};
P[2906]{
   GP1:
	UF : 0, UT : 6,		CONFIG : 'N U T, 0, 0, 0',
	X =  216.542  mm,	Y =   -612.809  mm,	Z =   -236.220  mm,
	W =  90.000 deg,	P =   0.000 deg,	R =   90.000 deg
};
P[2907]{
   GP1:
	UF : 0, UT : 6,		CONFIG : 'N U T, 0, 0, 0',
	X =  217.891  mm,	Y =   -611.930  mm,	Z =   -236.459  mm,
	W =  90.000 deg,	P =   0.000 deg,	R =   90.000 deg
};
P[2908]{
   GP1:
	UF : 0, UT : 6,		CONFIG : 'N U T, 0, 0, 0',
	X =  221.360  mm,	Y =   -610.020  mm,	Z =   -236.234  mm,
	W =  90.000 deg,	P =   0.000 deg,	R =   90.000 deg
};
P[2909]{
   GP1:
	UF : 0, UT : 6,		CONFIG : 'N U T, 0, 0, 0',
	X =  226.110  mm,	Y =   -607.227  mm,	Z =   -236.357  mm,
	W =  90.000 deg,	P =   0.000 deg,	R =   90.000 deg
};
P[2910]{
   GP1:
	UF : 0, UT : 6,		CONFIG : 'N U T, 0, 0, 0',
	X =  227.180  mm,	Y =   -606.559  mm,	Z =   -236.479  mm,
	W =  90.000 deg,	P =   0.000 deg,	R =   90.000 deg
};
P[2911]{
   GP1:
	UF : 0, UT : 6,		CONFIG : 'N U T, 0, 0, 0',
	X =  229.999  mm,	Y =   -604.949  mm,	Z =   -236.435  mm,
	W =  90.000 deg,	P =   0.000 deg,	R =   90.000 deg
};
P[2912]{
   GP1:
	UF : 0, UT : 6,		CONFIG : 'N U T, 0, 0, 0',
	X =  232.045  mm,	Y =   -603.803  mm,	Z =   -236.351  mm,
	W =  90.000 deg,	P =   0.000 deg,	R =   90.000 deg
};
P[2913]{
   GP1:
	UF : 0, UT : 6,		CONFIG : 'N U T, 0, 0, 0',
	X =  232.833  mm,	Y =   -603.352  mm,	Z =   -236.340  mm,
	W =  90.000 deg,	P =   0.000 deg,	R =   90.000 deg
};
P[2914]{
   GP1:
	UF : 0, UT : 6,		CONFIG : 'N U T, 0, 0, 0',
	X =  235.224  mm,	Y =   -602.044  mm,	Z =   -236.165  mm,
	W =  90.000 deg,	P =   0.000 deg,	R =   90.000 deg
};
P[2915]{
   GP1:
	UF : 0, UT : 6,		CONFIG : 'N U T, 0, 0, 0',
	X =  236.401  mm,	Y =   -601.273  mm,	Z =   -236.386  mm,
	W =  90.000 deg,	P =   0.000 deg,	R =   90.000 deg
};
P[2916]{
   GP1:
	UF : 0, UT : 6,		CONFIG : 'N U T, 0, 0, 0',
	X =  239.843  mm,	Y =   -599.277  mm,	Z =   -236.408  mm,
	W =  90.000 deg,	P =   0.000 deg,	R =   90.000 deg
};
P[2917]{
   GP1:
	UF : 0, UT : 6,		CONFIG : 'N U T, 0, 0, 0',
	X =  241.795  mm,	Y =   -598.204  mm,	Z =   -236.275  mm,
	W =  90.000 deg,	P =   0.000 deg,	R =   90.000 deg
};
P[2918]{
   GP1:
	UF : 0, UT : 6,		CONFIG : 'N U T, 0, 0, 0',
	X =  243.604  mm,	Y =   -597.089  mm,	Z =   -236.447  mm,
	W =  90.000 deg,	P =   0.000 deg,	R =   90.000 deg
};
P[2919]{
   GP1:
	UF : 0, UT : 6,		CONFIG : 'N U T, 0, 0, 0',
	X =  245.095  mm,	Y =   -596.240  mm,	Z =   -236.417  mm,
	W =  90.000 deg,	P =   0.000 deg,	R =   90.000 deg
};
P[2920]{
   GP1:
	UF : 0, UT : 6,		CONFIG : 'N U T, 0, 0, 0',
	X =  250.317  mm,	Y =   -593.255  mm,	Z =   -236.345  mm,
	W =  90.000 deg,	P =   0.000 deg,	R =   90.000 deg
};
P[2921]{
   GP1:
	UF : 0, UT : 6,		CONFIG : 'N U T, 0, 0, 0',
	X =  251.261  mm,	Y =   -592.838  mm,	Z =   -236.036  mm,
	W =  90.000 deg,	P =   0.000 deg,	R =   90.000 deg
};
P[2922]{
   GP1:
	UF : 0, UT : 6,		CONFIG : 'N U T, 0, 0, 0',
	X =  254.626  mm,	Y =   -590.767  mm,	Z =   -236.345  mm,
	W =  90.000 deg,	P =   0.000 deg,	R =   90.000 deg
};
P[2923]{
   GP1:
	UF : 0, UT : 6,		CONFIG : 'N U T, 0, 0, 0',
	X =  257.189  mm,	Y =   -589.366  mm,	Z =   -236.153  mm,
	W =  90.000 deg,	P =   0.000 deg,	R =   90.000 deg
};
P[2924]{
   GP1:
	UF : 0, UT : 6,		CONFIG : 'N U T, 0, 0, 0',
	X =  259.866  mm,	Y =   -587.702  mm,	Z =   -236.441  mm,
	W =  90.000 deg,	P =   0.000 deg,	R =   90.000 deg
};
P[2925]{
   GP1:
	UF : 0, UT : 6,		CONFIG : 'N U T, 0, 0, 0',
	X =  266.555  mm,	Y =   -583.821  mm,	Z =   -236.486  mm,
	W =  90.000 deg,	P =   0.000 deg,	R =   90.000 deg
};
P[2926]{
   GP1:
	UF : 0, UT : 6,		CONFIG : 'N U T, 0, 0, 0',
	X =  267.190  mm,	Y =   -583.617  mm,	Z =   -236.093  mm,
	W =  90.000 deg,	P =   0.000 deg,	R =   90.000 deg
};
P[2927]{
   GP1:
	UF : 0, UT : 6,		CONFIG : 'N U T, 0, 0, 0',
	X =  269.211  mm,	Y =   -582.413  mm,	Z =   -236.179  mm,
	W =  90.000 deg,	P =   0.000 deg,	R =   90.000 deg
};
P[2928]{
   GP1:
	UF : 0, UT : 6,		CONFIG : 'N U T, 0, 0, 0',
	X =  269.805  mm,	Y =   -581.994  mm,	Z =   -236.367  mm,
	W =  90.000 deg,	P =   0.000 deg,	R =   90.000 deg
};
P[2929]{
   GP1:
	UF : 0, UT : 6,		CONFIG : 'N U T, 0, 0, 0',
	X =  274.178  mm,	Y =   -579.470  mm,	Z =   -236.364  mm,
	W =  90.000 deg,	P =   0.000 deg,	R =   90.000 deg
};
P[2930]{
   GP1:
	UF : 0, UT : 6,		CONFIG : 'N U T, 0, 0, 0',
	X =  275.282  mm,	Y =   -578.863  mm,	Z =   -236.289  mm,
	W =  90.000 deg,	P =   0.000 deg,	R =   90.000 deg
};
P[2931]{
   GP1:
	UF : 0, UT : 6,		CONFIG : 'N U T, 0, 0, 0',
	X =  279.257  mm,	Y =   -576.664  mm,	Z =   -236.057  mm,
	W =  90.000 deg,	P =   0.000 deg,	R =   90.000 deg
};
P[2932]{
   GP1:
	UF : 0, UT : 6,		CONFIG : 'N U T, 0, 0, 0',
	X =  279.912  mm,	Y =   -576.167  mm,	Z =   -236.346  mm,
	W =  90.000 deg,	P =   0.000 deg,	R =   90.000 deg
};
P[2933]{
   GP1:
	UF : 0, UT : 6,		CONFIG : 'N U T, 0, 0, 0',
	X =  281.022  mm,	Y =   -575.649  mm,	Z =   -236.046  mm,
	W =  90.000 deg,	P =   0.000 deg,	R =   90.000 deg
};
P[2934]{
   GP1:
	UF : 0, UT : 6,		CONFIG : 'N U T, 0, 0, 0',
	X =  282.421  mm,	Y =   -574.808  mm,	Z =   -236.129  mm,
	W =  90.000 deg,	P =   0.000 deg,	R =   90.000 deg
};
P[2935]{
   GP1:
	UF : 0, UT : 6,		CONFIG : 'N U T, 0, 0, 0',
	X =  285.549  mm,	Y =   -572.962  mm,	Z =   -236.224  mm,
	W =  90.000 deg,	P =   0.000 deg,	R =   90.000 deg
};
P[2936]{
   GP1:
	UF : 0, UT : 6,		CONFIG : 'N U T, 0, 0, 0',
	X =  288.330  mm,	Y =   -571.299  mm,	Z =   -236.363  mm,
	W =  90.000 deg,	P =   0.000 deg,	R =   90.000 deg
};
P[2937]{
   GP1:
	UF : 0, UT : 6,		CONFIG : 'N U T, 0, 0, 0',
	X =  289.285  mm,	Y =   -570.792  mm,	Z =   -236.256  mm,
	W =  90.000 deg,	P =   0.000 deg,	R =   90.000 deg
};
P[2938]{
   GP1:
	UF : 0, UT : 6,		CONFIG : 'N U T, 0, 0, 0',
	X =  291.057  mm,	Y =   -569.670  mm,	Z =   -236.495  mm,
	W =  90.000 deg,	P =   0.000 deg,	R =   90.000 deg
};
P[2939]{
   GP1:
	UF : 0, UT : 6,		CONFIG : 'N U T, 0, 0, 0',
	X =  292.108  mm,	Y =   -569.173  mm,	Z =   -236.230  mm,
	W =  90.000 deg,	P =   0.000 deg,	R =   90.000 deg
};
P[2940]{
   GP1:
	UF : 0, UT : 6,		CONFIG : 'N U T, 0, 0, 0',
	X =  293.963  mm,	Y =   -568.165  mm,	Z =   -236.076  mm,
	W =  90.000 deg,	P =   0.000 deg,	R =   90.000 deg
};
P[2941]{
   GP1:
	UF : 0, UT : 6,		CONFIG : 'N U T, 0, 0, 0',
	X =  297.861  mm,	Y =   -565.756  mm,	Z =   -236.461  mm,
	W =  90.000 deg,	P =   0.000 deg,	R =   90.000 deg
};
P[2942]{
   GP1:
	UF : 0, UT : 6,		CONFIG : 'N U T, 0, 0, 0',
	X =  298.930  mm,	Y =   -565.134  mm,	Z =   -236.472  mm,
	W =  90.000 deg,	P =   0.000 deg,	R =   90.000 deg
};
P[2943]{
   GP1:
	UF : 0, UT : 6,		CONFIG : 'N U T, 0, 0, 0',
	X =  301.928  mm,	Y =   -563.428  mm,	Z =   -236.410  mm,
	W =  90.000 deg,	P =   0.000 deg,	R =   90.000 deg
};
P[2944]{
   GP1:
	UF : 0, UT : 6,		CONFIG : 'N U T, 0, 0, 0',
	X =  303.994  mm,	Y =   -562.195  mm,	Z =   -236.507  mm,
	W =  90.000 deg,	P =   0.000 deg,	R =   90.000 deg
};
P[2945]{
   GP1:
	UF : 0, UT : 6,		CONFIG : 'N U T, 0, 0, 0',
	X =  305.877  mm,	Y =   -561.200  mm,	Z =   -236.284  mm,
	W =  90.000 deg,	P =   0.000 deg,	R =   90.000 deg
};
P[2946]{
   GP1:
	UF : 0, UT : 6,		CONFIG : 'N U T, 0, 0, 0',
	X =  307.852  mm,	Y =   -560.132  mm,	Z =   -236.108  mm,
	W =  90.000 deg,	P =   0.000 deg,	R =   90.000 deg
};
P[2947]{
   GP1:
	UF : 0, UT : 6,		CONFIG : 'N U T, 0, 0, 0',
	X =  309.488  mm,	Y =   -559.059  mm,	Z =   -236.421  mm,
	W =  90.000 deg,	P =   0.000 deg,	R =   90.000 deg
};
P[2948]{
   GP1:
	UF : 0, UT : 6,		CONFIG : 'N U T, 0, 0, 0',
	X =  311.523  mm,	Y =   -557.908  mm,	Z =   -236.361  mm,
	W =  90.000 deg,	P =   0.000 deg,	R =   90.000 deg
};
P[2949]{
   GP1:
	UF : 0, UT : 6,		CONFIG : 'N U T, 0, 0, 0',
	X =  312.456  mm,	Y =   -557.349  mm,	Z =   -236.410  mm,
	W =  90.000 deg,	P =   0.000 deg,	R =   90.000 deg
};
P[2950]{
   GP1:
	UF : 0, UT : 6,		CONFIG : 'N U T, 0, 0, 0',
	X =  314.048  mm,	Y =   -556.527  mm,	Z =   -236.176  mm,
	W =  90.000 deg,	P =   0.000 deg,	R =   90.000 deg
};
P[2951]{
   GP1:
	UF : 0, UT : 6,		CONFIG : 'N U T, 0, 0, 0',
	X =  315.315  mm,	Y =   -555.701  mm,	Z =   -236.406  mm,
	W =  90.000 deg,	P =   0.000 deg,	R =   90.000 deg
};
P[2952]{
   GP1:
	UF : 0, UT : 6,		CONFIG : 'N U T, 0, 0, 0',
	X =  317.801  mm,	Y =   -554.401  mm,	Z =   -236.077  mm,
	W =  90.000 deg,	P =   0.000 deg,	R =   90.000 deg
};
P[2953]{
   GP1:
	UF : 0, UT : 6,		CONFIG : 'N U T, 0, 0, 0',
	X =  319.773  mm,	Y =   -553.120  mm,	Z =   -236.421  mm,
	W =  90.000 deg,	P =   0.000 deg,	R =   90.000 deg
};
P[2954]{
   GP1:
	UF : 0, UT : 6,		CONFIG : 'N U T, 0, 0, 0',
	X =  320.697  mm,	Y =   -552.561  mm,	Z =   -236.484  mm,
	W =  90.000 deg,	P =   0.000 deg,	R =   90.000 deg
};
P[2955]{
   GP1:
	UF : 0, UT : 6,		CONFIG : 'N U T, 0, 0, 0',
	X =  321.655  mm,	Y =   -552.016  mm,	Z =   -236.464  mm,
	W =  90.000 deg,	P =   0.000 deg,	R =   90.000 deg
};
P[2956]{
   GP1:
	UF : 0, UT : 6,		CONFIG : 'N U T, 0, 0, 0',
	X =  324.243  mm,	Y =   -550.616  mm,	Z =   -236.235  mm,
	W =  90.000 deg,	P =   0.000 deg,	R =   90.000 deg
};
P[2957]{
   GP1:
	UF : 0, UT : 6,		CONFIG : 'N U T, 0, 0, 0',
	X =  325.458  mm,	Y =   -549.839  mm,	Z =   -236.418  mm,
	W =  90.000 deg,	P =   0.000 deg,	R =   90.000 deg
};
P[2958]{
   GP1:
	UF : 0, UT : 6,		CONFIG : 'N U T, 0, 0, 0',
	X =  326.329  mm,	Y =   -549.397  mm,	Z =   -236.271  mm,
	W =  90.000 deg,	P =   0.000 deg,	R =   90.000 deg
};
P[2959]{
   GP1:
	UF : 0, UT : 6,		CONFIG : 'N U T, 0, 0, 0',
	X =  327.359  mm,	Y =   -548.901  mm,	Z =   -236.029  mm,
	W =  90.000 deg,	P =   0.000 deg,	R =   90.000 deg
};
P[2960]{
   GP1:
	UF : 0, UT : 6,		CONFIG : 'N U T, 0, 0, 0',
	X =  329.773  mm,	Y =   -547.339  mm,	Z =   -236.439  mm,
	W =  90.000 deg,	P =   0.000 deg,	R =   90.000 deg
};
P[2961]{
   GP1:
	UF : 0, UT : 6,		CONFIG : 'N U T, 0, 0, 0',
	X =  333.590  mm,	Y =   -545.228  mm,	Z =   -236.213  mm,
	W =  90.000 deg,	P =   0.000 deg,	R =   90.000 deg
};
P[2962]{
   GP1:
	UF : 0, UT : 6,		CONFIG : 'N U T, 0, 0, 0',
	X =  334.421  mm,	Y =   -544.656  mm,	Z =   -236.437  mm,
	W =  90.000 deg,	P =   0.000 deg,	R =   90.000 deg
};
P[2963]{
   GP1:
	UF : 0, UT : 6,		CONFIG : 'N U T, 0, 0, 0',
	X =  335.325  mm,	Y =   -544.222  mm,	Z =   -236.223  mm,
	W =  90.000 deg,	P =   0.000 deg,	R =   90.000 deg
};
P[2964]{
   GP1:
	UF : 0, UT : 6,		CONFIG : 'N U T, 0, 0, 0',
	X =  339.710  mm,	Y =   -541.730  mm,	Z =   -236.129  mm,
	W =  90.000 deg,	P =   0.000 deg,	R =   90.000 deg
};
P[2965]{
   GP1:
	UF : 0, UT : 6,		CONFIG : 'N U T, 0, 0, 0',
	X =  342.049  mm,	Y =   -540.362  mm,	Z =   -236.169  mm,
	W =  90.000 deg,	P =   0.000 deg,	R =   90.000 deg
};
P[2966]{
   GP1:
	UF : 0, UT : 6,		CONFIG : 'N U T, 0, 0, 0',
	X =  344.894  mm,	Y =   -538.651  mm,	Z =   -236.333  mm,
	W =  90.000 deg,	P =   0.000 deg,	R =   90.000 deg
};
P[2967]{
   GP1:
	UF : 0, UT : 6,		CONFIG : 'N U T, 0, 0, 0',
	X =  347.013  mm,	Y =   -537.494  mm,	Z =   -236.173  mm,
	W =  90.000 deg,	P =   0.000 deg,	R =   90.000 deg
};
P[2968]{
   GP1:
	UF : 0, UT : 6,		CONFIG : 'N U T, 0, 0, 0',
	X =  349.396  mm,	Y =   -536.107  mm,	Z =   -236.203  mm,
	W =  90.000 deg,	P =   0.000 deg,	R =   90.000 deg
};
P[2969]{
   GP1:
	UF : 0, UT : 6,		CONFIG : 'N U T, 0, 0, 0',
	X =  350.110  mm,	Y =   -535.604  mm,	Z =   -236.422  mm,
	W =  90.000 deg,	P =   0.000 deg,	R =   90.000 deg
};
P[2970]{
   GP1:
	UF : 0, UT : 6,		CONFIG : 'N U T, 0, 0, 0',
	X =  351.340  mm,	Y =   -534.959  mm,	Z =   -236.262  mm,
	W =  90.000 deg,	P =   0.000 deg,	R =   90.000 deg
};
P[2971]{
   GP1:
	UF : 0, UT : 6,		CONFIG : 'N U T, 0, 0, 0',
	X =  356.719  mm,	Y =   -531.822  mm,	Z =   -236.340  mm,
	W =  90.000 deg,	P =   0.000 deg,	R =   90.000 deg
};
P[2972]{
   GP1:
	UF : 0, UT : 6,		CONFIG : 'N U T, 0, 0, 0',
	X =  359.009  mm,	Y =   -530.563  mm,	Z =   -236.185  mm,
	W =  90.000 deg,	P =   0.000 deg,	R =   90.000 deg
};
P[2973]{
   GP1:
	UF : 0, UT : 6,		CONFIG : 'N U T, 0, 0, 0',
	X =  361.667  mm,	Y =   -529.048  mm,	Z =   -236.137  mm,
	W =  90.000 deg,	P =   0.000 deg,	R =   90.000 deg
};
P[2974]{
   GP1:
	UF : 0, UT : 6,		CONFIG : 'N U T, 0, 0, 0',
	X =  369.212  mm,	Y =   -524.580  mm,	Z =   -236.409  mm,
	W =  90.000 deg,	P =   0.000 deg,	R =   90.000 deg
};
P[2975]{
   GP1:
	UF : 0, UT : 6,		CONFIG : 'N U T, 0, 0, 0',
	X =  370.099  mm,	Y =   -524.029  mm,	Z =   -236.504  mm,
	W =  90.000 deg,	P =   0.000 deg,	R =   90.000 deg
};
P[2976]{
   GP1:
	UF : 0, UT : 6,		CONFIG : 'N U T, 0, 0, 0',
	X =  371.533  mm,	Y =   -523.242  mm,	Z =   -236.403  mm,
	W =  90.000 deg,	P =   0.000 deg,	R =   90.000 deg
};
P[2977]{
   GP1:
	UF : 0, UT : 6,		CONFIG : 'N U T, 0, 0, 0',
	X =  373.921  mm,	Y =   -521.948  mm,	Z =   -236.196  mm,
	W =  90.000 deg,	P =   0.000 deg,	R =   90.000 deg
};
P[2978]{
   GP1:
	UF : 0, UT : 6,		CONFIG : 'N U T, 0, 0, 0',
	X =  376.104  mm,	Y =   -520.695  mm,	Z =   -236.181  mm,
	W =  90.000 deg,	P =   0.000 deg,	R =   90.000 deg
};
P[2979]{
   GP1:
	UF : 0, UT : 6,		CONFIG : 'N U T, 0, 0, 0',
	X =  377.827  mm,	Y =   -519.584  mm,	Z =   -236.459  mm,
	W =  90.000 deg,	P =   0.000 deg,	R =   90.000 deg
};
P[2980]{
   GP1:
	UF : 0, UT : 6,		CONFIG : 'N U T, 0, 0, 0',
	X =  378.443  mm,	Y =   -519.360  mm,	Z =   -236.143  mm,
	W =  90.000 deg,	P =   0.000 deg,	R =   90.000 deg
};
P[2981]{
   GP1:
	UF : 0, UT : 6,		CONFIG : 'N U T, 0, 0, 0',
	X =  379.111  mm,	Y =   -518.915  mm,	Z =   -236.284  mm,
	W =  90.000 deg,	P =   0.000 deg,	R =   90.000 deg
};
P[2982]{
   GP1:
	UF : 0, UT : 6,		CONFIG : 'N U T, 0, 0, 0',
	X =  379.948  mm,	Y =   -518.418  mm,	Z =   -236.318  mm,
	W =  90.000 deg,	P =   0.000 deg,	R =   90.000 deg
};
P[2983]{
   GP1:
	UF : 0, UT : 6,		CONFIG : 'N U T, 0, 0, 0',
	X =  380.774  mm,	Y =   -517.964  mm,	Z =   -236.264  mm,
	W =  90.000 deg,	P =   0.000 deg,	R =   90.000 deg
};
P[2984]{
   GP1:
	UF : 0, UT : 6,		CONFIG : 'N U T, 0, 0, 0',
	X =  381.916  mm,	Y =   -517.290  mm,	Z =   -236.300  mm,
	W =  90.000 deg,	P =   0.000 deg,	R =   90.000 deg
};
P[2985]{
   GP1:
	UF : 0, UT : 6,		CONFIG : 'N U T, 0, 0, 0',
	X =  383.511  mm,	Y =   -516.342  mm,	Z =   -236.363  mm,
	W =  90.000 deg,	P =   0.000 deg,	R =   90.000 deg
};
P[2986]{
   GP1:
	UF : 0, UT : 6,		CONFIG : 'N U T, 0, 0, 0',
	X =  384.542  mm,	Y =   -515.853  mm,	Z =   -236.105  mm,
	W =  90.000 deg,	P =   0.000 deg,	R =   90.000 deg
};
P[2987]{
   GP1:
	UF : 0, UT : 6,		CONFIG : 'N U T, 0, 0, 0',
	X =  386.428  mm,	Y =   -514.621  mm,	Z =   -236.451  mm,
	W =  90.000 deg,	P =   0.000 deg,	R =   90.000 deg
};
P[2988]{
   GP1:
	UF : 0, UT : 6,		CONFIG : 'N U T, 0, 0, 0',
	X =  387.190  mm,	Y =   -514.184  mm,	Z =   -236.447  mm,
	W =  90.000 deg,	P =   0.000 deg,	R =   90.000 deg
};
P[2989]{
   GP1:
	UF : 0, UT : 6,		CONFIG : 'N U T, 0, 0, 0',
	X =  388.862  mm,	Y =   -513.326  mm,	Z =   -236.184  mm,
	W =  90.000 deg,	P =   0.000 deg,	R =   90.000 deg
};
P[2990]{
   GP1:
	UF : 0, UT : 6,		CONFIG : 'N U T, 0, 0, 0',
	X =  391.339  mm,	Y =   -511.857  mm,	Z =   -236.280  mm,
	W =  90.000 deg,	P =   0.000 deg,	R =   90.000 deg
};
P[2991]{
   GP1:
	UF : 0, UT : 6,		CONFIG : 'N U T, 0, 0, 0',
	X =  392.320  mm,	Y =   -511.373  mm,	Z =   -236.078  mm,
	W =  90.000 deg,	P =   0.000 deg,	R =   90.000 deg
};
P[2992]{
   GP1:
	UF : 0, UT : 6,		CONFIG : 'N U T, 0, 0, 0',
	X =  393.488  mm,	Y =   -510.523  mm,	Z =   -236.506  mm,
	W =  90.000 deg,	P =   0.000 deg,	R =   90.000 deg
};
P[2993]{
   GP1:
	UF : 0, UT : 6,		CONFIG : 'N U T, 0, 0, 0',
	X =  397.713  mm,	Y =   -508.084  mm,	Z =   -236.505  mm,
	W =  90.000 deg,	P =   0.000 deg,	R =   90.000 deg
};
P[2994]{
   GP1:
	UF : 0, UT : 6,		CONFIG : 'N U T, 0, 0, 0',
	X =  398.604  mm,	Y =   -507.575  mm,	Z =   -236.490  mm,
	W =  90.000 deg,	P =   0.000 deg,	R =   90.000 deg
};
P[2995]{
   GP1:
	UF : 0, UT : 6,		CONFIG : 'N U T, 0, 0, 0',
	X =  399.874  mm,	Y =   -506.914  mm,	Z =   -236.314  mm,
	W =  90.000 deg,	P =   0.000 deg,	R =   90.000 deg
};
P[2996]{
   GP1:
	UF : 0, UT : 6,		CONFIG : 'N U T, 0, 0, 0',
	X =  402.976  mm,	Y =   -505.077  mm,	Z =   -236.428  mm,
	W =  90.000 deg,	P =   0.000 deg,	R =   90.000 deg
};
P[2997]{
   GP1:
	UF : 0, UT : 6,		CONFIG : 'N U T, 0, 0, 0',
	X =  404.780  mm,	Y =   -504.061  mm,	Z =   -236.364  mm,
	W =  90.000 deg,	P =   0.000 deg,	R =   90.000 deg
};
P[2998]{
   GP1:
	UF : 0, UT : 6,		CONFIG : 'N U T, 0, 0, 0',
	X =  407.751  mm,	Y =   -502.447  mm,	Z =   -236.117  mm,
	W =  90.000 deg,	P =   0.000 deg,	R =   90.000 deg
};
P[2999]{
   GP1:
	UF : 0, UT : 6,		CONFIG : 'N U T, 0, 0, 0',
	X =  409.402  mm,	Y =   -501.371  mm,	Z =   -236.417  mm,
	W =  90.000 deg,	P =   0.000 deg,	R =   90.000 deg
};
P[3000]{
   GP1:
	UF : 0, UT : 6,		CONFIG : 'N U T, 0, 0, 0',
	X =  410.368  mm,	Y =   -500.890  mm,	Z =   -236.229  mm,
	W =  90.000 deg,	P =   0.000 deg,	R =   90.000 deg
};
P[3001]{
   GP1:
	UF : 0, UT : 6,		CONFIG : 'N U T, 0, 0, 0',
	X =  411.382  mm,	Y =   -500.370  mm,	Z =   -236.070  mm,
	W =  90.000 deg,	P =   0.000 deg,	R =   90.000 deg
};
P[3002]{
   GP1:
	UF : 0, UT : 6,		CONFIG : 'N U T, 0, 0, 0',
	X =  414.751  mm,	Y =   -498.290  mm,	Z =   -236.399  mm,
	W =  90.000 deg,	P =   0.000 deg,	R =   90.000 deg
};
P[3003]{
   GP1:
	UF : 0, UT : 6,		CONFIG : 'N U T, 0, 0, 0',
	X =  416.813  mm,	Y =   -497.205  mm,	Z =   -236.141  mm,
	W =  90.000 deg,	P =   0.000 deg,	R =   90.000 deg
};
P[3004]{
   GP1:
	UF : 0, UT : 6,		CONFIG : 'N U T, 0, 0, 0',
	X =  417.444  mm,	Y =   -496.735  mm,	Z =   -236.398  mm,
	W =  90.000 deg,	P =   0.000 deg,	R =   90.000 deg
};
P[3005]{
   GP1:
	UF : 0, UT : 6,		CONFIG : 'N U T, 0, 0, 0',
	X =  418.185  mm,	Y =   -496.457  mm,	Z =   -236.034  mm,
	W =  90.000 deg,	P =   0.000 deg,	R =   90.000 deg
};
P[3006]{
   GP1:
	UF : 0, UT : 6,		CONFIG : 'N U T, 0, 0, 0',
	X =  420.720  mm,	Y =   -494.817  mm,	Z =   -236.464  mm,
	W =  90.000 deg,	P =   0.000 deg,	R =   90.000 deg
};
P[3007]{
   GP1:
	UF : 0, UT : 6,		CONFIG : 'N U T, 0, 0, 0',
	X =  421.642  mm,	Y =   -494.294  mm,	Z =   -236.440  mm,
	W =  90.000 deg,	P =   0.000 deg,	R =   90.000 deg
};
P[3008]{
   GP1:
	UF : 0, UT : 6,		CONFIG : 'N U T, 0, 0, 0',
	X =  423.191  mm,	Y =   -493.476  mm,	Z =   -236.255  mm,
	W =  90.000 deg,	P =   0.000 deg,	R =   90.000 deg
};
P[3009]{
   GP1:
	UF : 0, UT : 6,		CONFIG : 'N U T, 0, 0, 0',
	X =  425.977  mm,	Y =   -491.880  mm,	Z =   -236.223  mm,
	W =  90.000 deg,	P =   0.000 deg,	R =   90.000 deg
};
P[3010]{
   GP1:
	UF : 0, UT : 6,		CONFIG : 'N U T, 0, 0, 0',
	X =  427.019  mm,	Y =   -491.205  mm,	Z =   -236.403  mm,
	W =  90.000 deg,	P =   0.000 deg,	R =   90.000 deg
};
P[3011]{
   GP1:
	UF : 0, UT : 6,		CONFIG : 'N U T, 0, 0, 0',
	X =  427.936  mm,	Y =   -490.657  mm,	Z =   -236.450  mm,
	W =  90.000 deg,	P =   0.000 deg,	R =   90.000 deg
};
P[3012]{
   GP1:
	UF : 0, UT : 6,		CONFIG : 'N U T, 0, 0, 0',
	X =  428.591  mm,	Y =   -490.284  mm,	Z =   -236.436  mm,
	W =  90.000 deg,	P =   0.000 deg,	R =   90.000 deg
};
P[3013]{
   GP1:
	UF : 0, UT : 6,		CONFIG : 'N U T, 0, 0, 0',
	X =  429.314  mm,	Y =   -489.884  mm,	Z =   -236.392  mm,
	W =  90.000 deg,	P =   0.000 deg,	R =   90.000 deg
};
P[3014]{
   GP1:
	UF : 0, UT : 6,		CONFIG : 'N U T, 0, 0, 0',
	X =  430.511  mm,	Y =   -489.291  mm,	Z =   -236.155  mm,
	W =  90.000 deg,	P =   0.000 deg,	R =   90.000 deg
};
P[3015]{
   GP1:
	UF : 0, UT : 6,		CONFIG : 'N U T, 0, 0, 0',
	X =  432.204  mm,	Y =   -488.192  mm,	Z =   -236.450  mm,
	W =  90.000 deg,	P =   0.000 deg,	R =   90.000 deg
};
P[3016]{
   GP1:
	UF : 0, UT : 6,		CONFIG : 'N U T, 0, 0, 0',
	X =  433.524  mm,	Y =   -487.432  mm,	Z =   -236.445  mm,
	W =  90.000 deg,	P =   0.000 deg,	R =   90.000 deg
};
P[3017]{
   GP1:
	UF : 0, UT : 6,		CONFIG : 'N U T, 0, 0, 0',
	X =  435.215  mm,	Y =   -486.570  mm,	Z =   -236.167  mm,
	W =  90.000 deg,	P =   0.000 deg,	R =   90.000 deg
};
P[3018]{
   GP1:
	UF : 0, UT : 6,		CONFIG : 'N U T, 0, 0, 0',
	X =  441.044  mm,	Y =   -483.085  mm,	Z =   -236.457  mm,
	W =  90.000 deg,	P =   0.000 deg,	R =   90.000 deg
};
P[3019]{
   GP1:
	UF : 0, UT : 6,		CONFIG : 'N U T, 0, 0, 0',
	X =  443.665  mm,	Y =   -481.699  mm,	Z =   -236.146  mm,
	W =  90.000 deg,	P =   0.000 deg,	R =   90.000 deg
};
P[3020]{
   GP1:
	UF : 0, UT : 6,		CONFIG : 'N U T, 0, 0, 0',
	X =  445.415  mm,	Y =   -480.673  mm,	Z =   -236.186  mm,
	W =  90.000 deg,	P =   0.000 deg,	R =   90.000 deg
};
P[3021]{
   GP1:
	UF : 0, UT : 6,		CONFIG : 'N U T, 0, 0, 0',
	X =  446.055  mm,	Y =   -480.240  mm,	Z =   -236.339  mm,
	W =  90.000 deg,	P =   0.000 deg,	R =   90.000 deg
};
P[3022]{
   GP1:
	UF : 0, UT : 6,		CONFIG : 'N U T, 0, 0, 0',
	X =  448.189  mm,	Y =   -478.996  mm,	Z =   -236.368  mm,
	W =  90.000 deg,	P =   0.000 deg,	R =   90.000 deg
};
P[3023]{
   GP1:
	UF : 0, UT : 6,		CONFIG : 'N U T, 0, 0, 0',
	X =  448.828  mm,	Y =   -478.629  mm,	Z =   -236.361  mm,
	W =  90.000 deg,	P =   0.000 deg,	R =   90.000 deg
};
P[3024]{
   GP1:
	UF : 0, UT : 6,		CONFIG : 'N U T, 0, 0, 0',
	X =  451.269  mm,	Y =   -477.179  mm,	Z =   -236.461  mm,
	W =  90.000 deg,	P =   0.000 deg,	R =   90.000 deg
};
P[3025]{
   GP1:
	UF : 0, UT : 6,		CONFIG : 'N U T, 0, 0, 0',
	X =  452.416  mm,	Y =   -476.598  mm,	Z =   -236.264  mm,
	W =  90.000 deg,	P =   0.000 deg,	R =   90.000 deg
};
P[3026]{
   GP1:
	UF : 0, UT : 6,		CONFIG : 'N U T, 0, 0, 0',
	X =  453.766  mm,	Y =   -475.879  mm,	Z =   -236.119  mm,
	W =  90.000 deg,	P =   0.000 deg,	R =   90.000 deg
};
P[3027]{
   GP1:
	UF : 0, UT : 6,		CONFIG : 'N U T, 0, 0, 0',
	X =  457.321  mm,	Y =   -473.766  mm,	Z =   -236.264  mm,
	W =  90.000 deg,	P =   0.000 deg,	R =   90.000 deg
};
P[3028]{
   GP1:
	UF : 0, UT : 6,		CONFIG : 'N U T, 0, 0, 0',
	X =  459.152  mm,	Y =   -472.669  mm,	Z =   -236.359  mm,
	W =  90.000 deg,	P =   0.000 deg,	R =   90.000 deg
};
P[3029]{
   GP1:
	UF : 0, UT : 6,		CONFIG : 'N U T, 0, 0, 0',
	X =  461.461  mm,	Y =   -471.304  mm,	Z =   -236.440  mm,
	W =  90.000 deg,	P =   0.000 deg,	R =   90.000 deg
};
P[3030]{
   GP1:
	UF : 0, UT : 6,		CONFIG : 'N U T, 0, 0, 0',
	X =  463.394  mm,	Y =   -470.358  mm,	Z =   -236.023  mm,
	W =  90.000 deg,	P =   0.000 deg,	R =   90.000 deg
};
P[3031]{
   GP1:
	UF : 0, UT : 6,		CONFIG : 'N U T, 0, 0, 0',
	X =  464.632  mm,	Y =   -469.478  mm,	Z =   -236.424  mm,
	W =  90.000 deg,	P =   0.000 deg,	R =   90.000 deg
};
P[3032]{
   GP1:
	UF : 0, UT : 6,		CONFIG : 'N U T, 0, 0, 0',
	X =  465.613  mm,	Y =   -468.911  mm,	Z =   -236.425  mm,
	W =  90.000 deg,	P =   0.000 deg,	R =   90.000 deg
};
P[3033]{
   GP1:
	UF : 0, UT : 6,		CONFIG : 'N U T, 0, 0, 0',
	X =  469.619  mm,	Y =   -466.625  mm,	Z =   -236.361  mm,
	W =  90.000 deg,	P =   0.000 deg,	R =   90.000 deg
};
P[3034]{
   GP1:
	UF : 0, UT : 6,		CONFIG : 'N U T, 0, 0, 0',
	X =  470.554  mm,	Y =   -466.183  mm,	Z =   -236.124  mm,
	W =  90.000 deg,	P =   0.000 deg,	R =   90.000 deg
};
P[3035]{
   GP1:
	UF : 0, UT : 6,		CONFIG : 'N U T, 0, 0, 0',
	X =  471.742  mm,	Y =   -465.379  mm,	Z =   -236.410  mm,
	W =  90.000 deg,	P =   0.000 deg,	R =   90.000 deg
};
P[3036]{
   GP1:
	UF : 0, UT : 6,		CONFIG : 'N U T, 0, 0, 0',
	X =  474.127  mm,	Y =   -463.992  mm,	Z =   -236.434  mm,
	W =  90.000 deg,	P =   0.000 deg,	R =   90.000 deg
};
P[3037]{
   GP1:
	UF : 0, UT : 6,		CONFIG : 'N U T, 0, 0, 0',
	X =  475.843  mm,	Y =   -462.993  mm,	Z =   -236.453  mm,
	W =  90.000 deg,	P =   0.000 deg,	R =   90.000 deg
};
P[3038]{
   GP1:
	UF : 0, UT : 6,		CONFIG : 'N U T, 0, 0, 0',
	X =  476.774  mm,	Y =   -462.542  mm,	Z =   -236.244  mm,
	W =  90.000 deg,	P =   0.000 deg,	R =   90.000 deg
};
P[3039]{
   GP1:
	UF : 0, UT : 6,		CONFIG : 'N U T, 0, 0, 0',
	X =  478.019  mm,	Y =   -461.806  mm,	Z =   -236.288  mm,
	W =  90.000 deg,	P =   0.000 deg,	R =   90.000 deg
};
P[3040]{
   GP1:
	UF : 0, UT : 6,		CONFIG : 'N U T, 0, 0, 0',
	X =  479.155  mm,	Y =   -461.075  mm,	Z =   -236.470  mm,
	W =  90.000 deg,	P =   0.000 deg,	R =   90.000 deg
};
P[3041]{
   GP1:
	UF : 0, UT : 6,		CONFIG : 'N U T, 0, 0, 0',
	X =  480.329  mm,	Y =   -460.470  mm,	Z =   -236.290  mm,
	W =  90.000 deg,	P =   0.000 deg,	R =   90.000 deg
};
P[3042]{
   GP1:
	UF : 0, UT : 6,		CONFIG : 'N U T, 0, 0, 0',
	X =  481.759  mm,	Y =   -459.600  mm,	Z =   -236.401  mm,
	W =  90.000 deg,	P =   0.000 deg,	R =   90.000 deg
};
P[3043]{
   GP1:
	UF : 0, UT : 6,		CONFIG : 'N U T, 0, 0, 0',
	X =  483.263  mm,	Y =   -458.745  mm,	Z =   -236.367  mm,
	W =  90.000 deg,	P =   0.000 deg,	R =   90.000 deg
};
P[3044]{
   GP1:
	UF : 0, UT : 6,		CONFIG : 'N U T, 0, 0, 0',
	X =  488.030  mm,	Y =   -455.938  mm,	Z =   -236.499  mm,
	W =  90.000 deg,	P =   0.000 deg,	R =   90.000 deg
};
P[3045]{
   GP1:
	UF : 0, UT : 6,		CONFIG : 'N U T, 0, 0, 0',
	X =  489.449  mm,	Y =   -455.233  mm,	Z =   -236.222  mm,
	W =  90.000 deg,	P =   0.000 deg,	R =   90.000 deg
};
P[3046]{
   GP1:
	UF : 0, UT : 6,		CONFIG : 'N U T, 0, 0, 0',
	X =  492.671  mm,	Y =   -453.340  mm,	Z =   -236.301  mm,
	W =  90.000 deg,	P =   0.000 deg,	R =   90.000 deg
};
P[3047]{
   GP1:
	UF : 0, UT : 6,		CONFIG : 'N U T, 0, 0, 0',
	X =  493.421  mm,	Y =   -452.952  mm,	Z =   -236.191  mm,
	W =  90.000 deg,	P =   0.000 deg,	R =   90.000 deg
};
P[3048]{
   GP1:
	UF : 0, UT : 6,		CONFIG : 'N U T, 0, 0, 0',
	X =  494.227  mm,	Y =   -452.449  mm,	Z =   -236.282  mm,
	W =  90.000 deg,	P =   0.000 deg,	R =   90.000 deg
};
P[3049]{
   GP1:
	UF : 0, UT : 6,		CONFIG : 'N U T, 0, 0, 0',
	X =  497.965  mm,	Y =   -450.288  mm,	Z =   -236.289  mm,
	W =  90.000 deg,	P =   0.000 deg,	R =   90.000 deg
};
P[3050]{
   GP1:
	UF : 0, UT : 6,		CONFIG : 'N U T, 0, 0, 0',
	X =  499.505  mm,	Y =   -449.309  mm,	Z =   -236.508  mm,
	W =  90.000 deg,	P =   0.000 deg,	R =   90.000 deg
};
P[3051]{
   GP1:
	UF : 0, UT : 6,		CONFIG : 'N U T, 0, 0, 0',
	X =  500.860  mm,	Y =   -448.561  mm,	Z =   -236.425  mm,
	W =  90.000 deg,	P =   0.000 deg,	R =   90.000 deg
};
P[3052]{
   GP1:
	UF : 0, UT : 6,		CONFIG : 'N U T, 0, 0, 0',
	X =  501.842  mm,	Y =   -447.975  mm,	Z =   -236.468  mm,
	W =  90.000 deg,	P =   0.000 deg,	R =   90.000 deg
};
P[3053]{
   GP1:
	UF : 0, UT : 6,		CONFIG : 'N U T, 0, 0, 0',
	X =  504.969  mm,	Y =   -446.168  mm,	Z =   -236.475  mm,
	W =  90.000 deg,	P =   0.000 deg,	R =   90.000 deg
};
P[3054]{
   GP1:
	UF : 0, UT : 6,		CONFIG : 'N U T, 0, 0, 0',
	X =  506.150  mm,	Y =   -445.637  mm,	Z =   -236.106  mm,
	W =  90.000 deg,	P =   0.000 deg,	R =   90.000 deg
};
P[3055]{
   GP1:
	UF : 0, UT : 6,		CONFIG : 'N U T, 0, 0, 0',
	X =  508.861  mm,	Y =   -443.907  mm,	Z =   -236.506  mm,
	W =  90.000 deg,	P =   0.000 deg,	R =   90.000 deg
};
P[3056]{
   GP1:
	UF : 0, UT : 6,		CONFIG : 'N U T, 0, 0, 0',
	X =  510.496  mm,	Y =   -442.979  mm,	Z =   -236.467  mm,
	W =  90.000 deg,	P =   0.000 deg,	R =   90.000 deg
};
P[3057]{
   GP1:
	UF : 0, UT : 6,		CONFIG : 'N U T, 0, 0, 0',
	X =  511.372  mm,	Y =   -442.576  mm,	Z =   -236.218  mm,
	W =  90.000 deg,	P =   0.000 deg,	R =   90.000 deg
};
P[3058]{
   GP1:
	UF : 0, UT : 6,		CONFIG : 'N U T, 0, 0, 0',
	X =  513.212  mm,	Y =   -441.486  mm,	Z =   -236.287  mm,
	W =  90.000 deg,	P =   0.000 deg,	R =   90.000 deg
};
P[3059]{
   GP1:
	UF : 0, UT : 6,		CONFIG : 'N U T, 0, 0, 0',
	X =  515.453  mm,	Y =   -440.128  mm,	Z =   -236.441  mm,
	W =  90.000 deg,	P =   0.000 deg,	R =   90.000 deg
};
P[3060]{
   GP1:
	UF : 0, UT : 6,		CONFIG : 'N U T, 0, 0, 0',
	X =  516.631  mm,	Y =   -439.469  mm,	Z =   -236.389  mm,
	W =  90.000 deg,	P =   0.000 deg,	R =   90.000 deg
};
P[3061]{
   GP1:
	UF : 0, UT : 6,		CONFIG : 'N U T, 0, 0, 0',
	X =  518.209  mm,	Y =   -438.567  mm,	Z =   -236.367  mm,
	W =  90.000 deg,	P =   0.000 deg,	R =   90.000 deg
};
P[3062]{
   GP1:
	UF : 0, UT : 6,		CONFIG : 'N U T, 0, 0, 0',
	X =  519.147  mm,	Y =   -438.019  mm,	Z =   -236.382  mm,
	W =  90.000 deg,	P =   0.000 deg,	R =   90.000 deg
};
P[3063]{
   GP1:
	UF : 0, UT : 6,		CONFIG : 'N U T, 0, 0, 0',
	X =  520.717  mm,	Y =   -437.060  mm,	Z =   -236.510  mm,
	W =  90.000 deg,	P =   0.000 deg,	R =   90.000 deg
};
P[3064]{
   GP1:
	UF : 0, UT : 6,		CONFIG : 'N U T, 0, 0, 0',
	X =  522.605  mm,	Y =   -435.992  mm,	Z =   -236.373  mm,
	W =  90.000 deg,	P =   0.000 deg,	R =   90.000 deg
};
P[3065]{
   GP1:
	UF : 0, UT : 6,		CONFIG : 'N U T, 0, 0, 0',
	X =  523.669  mm,	Y =   -435.352  mm,	Z =   -236.133  mm,
	W =  90.000 deg,	P =   0.000 deg,	R =   90.000 deg
};
P[3066]{
   GP1:
	UF : 0, UT : 6,		CONFIG : 'N U T, 0, 0, 0',
	X =  526.356  mm,	Y =   -432.681  mm,	Z =   -236.457  mm,
	W =  90.000 deg,	P =   0.000 deg,	R =   90.000 deg
};
P[3067]{
   GP1:
	UF : 0, UT : 6,		CONFIG : 'N U T, 0, 0, 0',
	X =  527.359  mm,	Y =   -431.504  mm,	Z =   -236.110  mm,
	W =  90.000 deg,	P =   0.000 deg,	R =   90.000 deg
};
P[3068]{
   GP1:
	UF : 0, UT : 6,		CONFIG : 'N U T, 0, 0, 0',
	X =  529.419  mm,	Y =   -425.700  mm,	Z =   -236.051  mm,
	W =  90.000 deg,	P =   0.000 deg,	R =   90.000 deg
};
P[3069]{
   GP1:
	UF : 0, UT : 6,		CONFIG : 'N U T, 0, 0, 0',
	X =  529.210  mm,	Y =   -422.774  mm,	Z =   -236.424  mm,
	W =  90.000 deg,	P =   0.000 deg,	R =   90.000 deg
};
P[3070]{
   GP1:
	UF : 0, UT : 6,		CONFIG : 'N U T, 0, 0, 0',
	X =  529.219  mm,	Y =   -421.939  mm,	Z =   -236.077  mm,
	W =  90.000 deg,	P =   0.000 deg,	R =   90.000 deg
};
P[3071]{
   GP1:
	UF : 0, UT : 6,		CONFIG : 'N U T, 0, 0, 0',
	X =  528.614  mm,	Y =   -420.021  mm,	Z =   -236.373  mm,
	W =  90.000 deg,	P =   0.000 deg,	R =   90.000 deg
};
P[3072]{
   GP1:
	UF : 0, UT : 6,		CONFIG : 'N U T, 0, 0, 0',
	X =  527.654  mm,	Y =   -417.928  mm,	Z =   -236.446  mm,
	W =  90.000 deg,	P =   0.000 deg,	R =   90.000 deg
};
P[3073]{
   GP1:
	UF : 0, UT : 6,		CONFIG : 'N U T, 0, 0, 0',
	X =  527.292  mm,	Y =   -417.200  mm,	Z =   -236.477  mm,
	W =  90.000 deg,	P =   0.000 deg,	R =   90.000 deg
};
P[3074]{
   GP1:
	UF : 0, UT : 6,		CONFIG : 'N U T, 0, 0, 0',
	X =  526.377  mm,	Y =   -415.574  mm,	Z =   -236.429  mm,
	W =  90.000 deg,	P =   0.000 deg,	R =   90.000 deg
};
P[3075]{
   GP1:
	UF : 0, UT : 6,		CONFIG : 'N U T, 0, 0, 0',
	X =  525.542  mm,	Y =   -414.103  mm,	Z =   -236.395  mm,
	W =  90.000 deg,	P =   0.000 deg,	R =   90.000 deg
};
P[3076]{
   GP1:
	UF : 0, UT : 6,		CONFIG : 'N U T, 0, 0, 0',
	X =  524.905  mm,	Y =   -412.881  mm,	Z =   -236.228  mm,
	W =  90.000 deg,	P =   0.000 deg,	R =   90.000 deg
};
P[3077]{
   GP1:
	UF : 0, UT : 6,		CONFIG : 'N U T, 0, 0, 0',
	X =  523.657  mm,	Y =   -410.911  mm,	Z =   -236.496  mm,
	W =  90.000 deg,	P =   0.000 deg,	R =   90.000 deg
};
P[3078]{
   GP1:
	UF : 0, UT : 6,		CONFIG : 'N U T, 0, 0, 0',
	X =  522.641  mm,	Y =   -409.147  mm,	Z =   -236.489  mm,
	W =  90.000 deg,	P =   0.000 deg,	R =   90.000 deg
};
P[3079]{
   GP1:
	UF : 0, UT : 6,		CONFIG : 'N U T, 0, 0, 0',
	X =  522.289  mm,	Y =   -408.340  mm,	Z =   -236.214  mm,
	W =  90.000 deg,	P =   0.000 deg,	R =   90.000 deg
};
P[3080]{
   GP1:
	UF : 0, UT : 6,		CONFIG : 'N U T, 0, 0, 0',
	X =  521.597  mm,	Y =   -407.331  mm,	Z =   -236.478  mm,
	W =  90.000 deg,	P =   0.000 deg,	R =   90.000 deg
};
P[3081]{
   GP1:
	UF : 0, UT : 6,		CONFIG : 'N U T, 0, 0, 0',
	X =  521.015  mm,	Y =   -406.291  mm,	Z =   -236.434  mm,
	W =  90.000 deg,	P =   0.000 deg,	R =   90.000 deg
};
P[3082]{
   GP1:
	UF : 0, UT : 6,		CONFIG : 'N U T, 0, 0, 0',
	X =  520.632  mm,	Y =   -405.382  mm,	Z =   -236.090  mm,
	W =  90.000 deg,	P =   0.000 deg,	R =   90.000 deg
};
P[3083]{
   GP1:
	UF : 0, UT : 6,		CONFIG : 'N U T, 0, 0, 0',
	X =  519.528  mm,	Y =   -403.674  mm,	Z =   -236.375  mm,
	W =  90.000 deg,	P =   0.000 deg,	R =   90.000 deg
};
P[3084]{
   GP1:
	UF : 0, UT : 6,		CONFIG : 'N U T, 0, 0, 0',
	X =  518.991  mm,	Y =   -402.654  mm,	Z =   -236.248  mm,
	W =  90.000 deg,	P =   0.000 deg,	R =   90.000 deg
};
P[3085]{
   GP1:
	UF : 0, UT : 6,		CONFIG : 'N U T, 0, 0, 0',
	X =  518.554  mm,	Y =   -402.039  mm,	Z =   -236.450  mm,
	W =  90.000 deg,	P =   0.000 deg,	R =   90.000 deg
};
P[3086]{
   GP1:
	UF : 0, UT : 6,		CONFIG : 'N U T, 0, 0, 0',
	X =  518.281  mm,	Y =   -401.278  mm,	Z =   -236.043  mm,
	W =  90.000 deg,	P =   0.000 deg,	R =   90.000 deg
};
P[3087]{
   GP1:
	UF : 0, UT : 6,		CONFIG : 'N U T, 0, 0, 0',
	X =  517.576  mm,	Y =   -400.372  mm,	Z =   -236.485  mm,
	W =  90.000 deg,	P =   0.000 deg,	R =   90.000 deg
};
P[3088]{
   GP1:
	UF : 0, UT : 6,		CONFIG : 'N U T, 0, 0, 0',
	X =  517.156  mm,	Y =   -399.342  mm,	Z =   -236.064  mm,
	W =  90.000 deg,	P =   0.000 deg,	R =   90.000 deg
};
P[3089]{
   GP1:
	UF : 0, UT : 6,		CONFIG : 'N U T, 0, 0, 0',
	X =  516.140  mm,	Y =   -397.832  mm,	Z =   -236.413  mm,
	W =  90.000 deg,	P =   0.000 deg,	R =   90.000 deg
};
P[3090]{
   GP1:
	UF : 0, UT : 6,		CONFIG : 'N U T, 0, 0, 0',
	X =  515.285  mm,	Y =   -396.147  mm,	Z =   -236.126  mm,
	W =  90.000 deg,	P =   0.000 deg,	R =   90.000 deg
};
P[3091]{
   GP1:
	UF : 0, UT : 6,		CONFIG : 'N U T, 0, 0, 0',
	X =  514.220  mm,	Y =   -394.340  mm,	Z =   -236.178  mm,
	W =  90.000 deg,	P =   0.000 deg,	R =   90.000 deg
};
P[3092]{
   GP1:
	UF : 0, UT : 6,		CONFIG : 'N U T, 0, 0, 0',
	X =  513.824  mm,	Y =   -393.765  mm,	Z =   -236.334  mm,
	W =  90.000 deg,	P =   0.000 deg,	R =   90.000 deg
};
P[3093]{
   GP1:
	UF : 0, UT : 6,		CONFIG : 'N U T, 0, 0, 0',
	X =  512.293  mm,	Y =   -391.222  mm,	Z =   -236.483  mm,
	W =  90.000 deg,	P =   0.000 deg,	R =   90.000 deg
};
P[3094]{
   GP1:
	UF : 0, UT : 6,		CONFIG : 'N U T, 0, 0, 0',
	X =  511.452  mm,	Y =   -389.757  mm,	Z =   -236.473  mm,
	W =  90.000 deg,	P =   0.000 deg,	R =   90.000 deg
};
P[3095]{
   GP1:
	UF : 0, UT : 6,		CONFIG : 'N U T, 0, 0, 0',
	X =  509.805  mm,	Y =   -386.908  mm,	Z =   -236.479  mm,
	W =  90.000 deg,	P =   0.000 deg,	R =   90.000 deg
};
P[3096]{
   GP1:
	UF : 0, UT : 6,		CONFIG : 'N U T, 0, 0, 0',
	X =  508.808  mm,	Y =   -384.934  mm,	Z =   -236.131  mm,
	W =  90.000 deg,	P =   0.000 deg,	R =   90.000 deg
};
P[3097]{
   GP1:
	UF : 0, UT : 6,		CONFIG : 'N U T, 0, 0, 0',
	X =  506.287  mm,	Y =   -380.723  mm,	Z =   -236.352  mm,
	W =  90.000 deg,	P =   0.000 deg,	R =   90.000 deg
};
P[3098]{
   GP1:
	UF : 0, UT : 6,		CONFIG : 'N U T, 0, 0, 0',
	X =  504.040  mm,	Y =   -376.934  mm,	Z =   -236.494  mm,
	W =  90.000 deg,	P =   0.000 deg,	R =   90.000 deg
};
P[3099]{
   GP1:
	UF : 0, UT : 6,		CONFIG : 'N U T, 0, 0, 0',
	X =  502.885  mm,	Y =   -374.840  mm,	Z =   -236.360  mm,
	W =  90.000 deg,	P =   0.000 deg,	R =   90.000 deg
};
P[3100]{
   GP1:
	UF : 0, UT : 6,		CONFIG : 'N U T, 0, 0, 0',
	X =  502.062  mm,	Y =   -373.465  mm,	Z =   -236.432  mm,
	W =  90.000 deg,	P =   0.000 deg,	R =   90.000 deg
};
P[3101]{
   GP1:
	UF : 0, UT : 6,		CONFIG : 'N U T, 0, 0, 0',
	X =  501.343  mm,	Y =   -372.194  mm,	Z =   -236.397  mm,
	W =  90.000 deg,	P =   0.000 deg,	R =   90.000 deg
};
P[3102]{
   GP1:
	UF : 0, UT : 6,		CONFIG : 'N U T, 0, 0, 0',
	X =  500.785  mm,	Y =   -371.305  mm,	Z =   -236.503  mm,
	W =  90.000 deg,	P =   0.000 deg,	R =   90.000 deg
};
P[3103]{
   GP1:
	UF : 0, UT : 6,		CONFIG : 'N U T, 0, 0, 0',
	X =  498.732  mm,	Y =   -367.699  mm,	Z =   -236.434  mm,
	W =  90.000 deg,	P =   0.000 deg,	R =   90.000 deg
};
P[3104]{
   GP1:
	UF : 0, UT : 6,		CONFIG : 'N U T, 0, 0, 0',
	X =  498.231  mm,	Y =   -366.885  mm,	Z =   -236.510  mm,
	W =  90.000 deg,	P =   0.000 deg,	R =   90.000 deg
};
P[3105]{
   GP1:
	UF : 0, UT : 6,		CONFIG : 'N U T, 0, 0, 0',
	X =  497.651  mm,	Y =   -365.620  mm,	Z =   -236.146  mm,
	W =  90.000 deg,	P =   0.000 deg,	R =   90.000 deg
};
P[3106]{
   GP1:
	UF : 0, UT : 6,		CONFIG : 'N U T, 0, 0, 0',
	X =  496.522  mm,	Y =   -363.886  mm,	Z =   -236.455  mm,
	W =  90.000 deg,	P =   0.000 deg,	R =   90.000 deg
};
P[3107]{
   GP1:
	UF : 0, UT : 6,		CONFIG : 'N U T, 0, 0, 0',
	X =  491.835  mm,	Y =   -355.669  mm,	Z =   -236.314  mm,
	W =  90.000 deg,	P =   0.000 deg,	R =   90.000 deg
};
P[3108]{
   GP1:
	UF : 0, UT : 6,		CONFIG : 'N U T, 0, 0, 0',
	X =  489.012  mm,	Y =   -350.676  mm,	Z =   -236.171  mm,
	W =  90.000 deg,	P =   0.000 deg,	R =   90.000 deg
};
P[3109]{
   GP1:
	UF : 0, UT : 6,		CONFIG : 'N U T, 0, 0, 0',
	X =  487.975  mm,	Y =   -348.842  mm,	Z =   -236.117  mm,
	W =  90.000 deg,	P =   0.000 deg,	R =   90.000 deg
};
P[3110]{
   GP1:
	UF : 0, UT : 6,		CONFIG : 'N U T, 0, 0, 0',
	X =  486.058  mm,	Y =   -345.599  mm,	Z =   -236.225  mm,
	W =  90.000 deg,	P =   0.000 deg,	R =   90.000 deg
};
P[3111]{
   GP1:
	UF : 0, UT : 6,		CONFIG : 'N U T, 0, 0, 0',
	X =  485.417  mm,	Y =   -344.654  mm,	Z =   -236.457  mm,
	W =  90.000 deg,	P =   0.000 deg,	R =   90.000 deg
};
P[3112]{
   GP1:
	UF : 0, UT : 6,		CONFIG : 'N U T, 0, 0, 0',
	X =  485.151  mm,	Y =   -343.954  mm,	Z =   -236.119  mm,
	W =  90.000 deg,	P =   0.000 deg,	R =   90.000 deg
};
P[3113]{
   GP1:
	UF : 0, UT : 6,		CONFIG : 'N U T, 0, 0, 0',
	X =  484.586  mm,	Y =   -343.229  mm,	Z =   -236.477  mm,
	W =  90.000 deg,	P =   0.000 deg,	R =   90.000 deg
};
P[3114]{
   GP1:
	UF : 0, UT : 6,		CONFIG : 'N U T, 0, 0, 0',
	X =  483.516  mm,	Y =   -341.282  mm,	Z =   -236.345  mm,
	W =  90.000 deg,	P =   0.000 deg,	R =   90.000 deg
};
P[3115]{
   GP1:
	UF : 0, UT : 6,		CONFIG : 'N U T, 0, 0, 0',
	X =  481.833  mm,	Y =   -338.362  mm,	Z =   -236.338  mm,
	W =  90.000 deg,	P =   0.000 deg,	R =   90.000 deg
};
P[3116]{
   GP1:
	UF : 0, UT : 6,		CONFIG : 'N U T, 0, 0, 0',
	X =  481.007  mm,	Y =   -336.999  mm,	Z =   -236.431  mm,
	W =  90.000 deg,	P =   0.000 deg,	R =   90.000 deg
};
P[3117]{
   GP1:
	UF : 0, UT : 6,		CONFIG : 'N U T, 0, 0, 0',
	X =  480.500  mm,	Y =   -336.121  mm,	Z =   -236.432  mm,
	W =  90.000 deg,	P =   0.000 deg,	R =   90.000 deg
};
P[3118]{
   GP1:
	UF : 0, UT : 6,		CONFIG : 'N U T, 0, 0, 0',
	X =  478.047  mm,	Y =   -331.828  mm,	Z =   -236.368  mm,
	W =  90.000 deg,	P =   0.000 deg,	R =   90.000 deg
};
P[3119]{
   GP1:
	UF : 0, UT : 6,		CONFIG : 'N U T, 0, 0, 0',
	X =  477.096  mm,	Y =   -330.183  mm,	Z =   -236.374  mm,
	W =  90.000 deg,	P =   0.000 deg,	R =   90.000 deg
};
P[3120]{
   GP1:
	UF : 0, UT : 6,		CONFIG : 'N U T, 0, 0, 0',
	X =  476.551  mm,	Y =   -329.315  mm,	Z =   -236.480  mm,
	W =  90.000 deg,	P =   0.000 deg,	R =   90.000 deg
};
P[3121]{
   GP1:
	UF : 0, UT : 6,		CONFIG : 'N U T, 0, 0, 0',
	X =  475.912  mm,	Y =   -328.159  mm,	Z =   -236.411  mm,
	W =  90.000 deg,	P =   0.000 deg,	R =   90.000 deg
};
P[3122]{
   GP1:
	UF : 0, UT : 6,		CONFIG : 'N U T, 0, 0, 0',
	X =  475.126  mm,	Y =   -326.776  mm,	Z =   -236.380  mm,
	W =  90.000 deg,	P =   0.000 deg,	R =   90.000 deg
};
P[3123]{
   GP1:
	UF : 0, UT : 6,		CONFIG : 'N U T, 0, 0, 0',
	X =  474.521  mm,	Y =   -325.697  mm,	Z =   -236.335  mm,
	W =  90.000 deg,	P =   0.000 deg,	R =   90.000 deg
};
P[3124]{
   GP1:
	UF : 0, UT : 6,		CONFIG : 'N U T, 0, 0, 0',
	X =  474.032  mm,	Y =   -324.909  mm,	Z =   -236.418  mm,
	W =  90.000 deg,	P =   0.000 deg,	R =   90.000 deg
};
P[3125]{
   GP1:
	UF : 0, UT : 6,		CONFIG : 'N U T, 0, 0, 0',
	X =  473.626  mm,	Y =   -323.924  mm,	Z =   -236.026  mm,
	W =  90.000 deg,	P =   0.000 deg,	R =   90.000 deg
};
P[3126]{
   GP1:
	UF : 0, UT : 6,		CONFIG : 'N U T, 0, 0, 0',
	X =  472.655  mm,	Y =   -322.587  mm,	Z =   -236.506  mm,
	W =  90.000 deg,	P =   0.000 deg,	R =   90.000 deg
};
P[3127]{
   GP1:
	UF : 0, UT : 6,		CONFIG : 'N U T, 0, 0, 0',
	X =  471.801  mm,	Y =   -320.902  mm,	Z =   -236.219  mm,
	W =  90.000 deg,	P =   0.000 deg,	R =   90.000 deg
};
P[3128]{
   GP1:
	UF : 0, UT : 6,		CONFIG : 'N U T, 0, 0, 0',
	X =  470.515  mm,	Y =   -318.794  mm,	Z =   -236.384  mm,
	W =  90.000 deg,	P =   0.000 deg,	R =   90.000 deg
};
P[3129]{
   GP1:
	UF : 0, UT : 6,		CONFIG : 'N U T, 0, 0, 0',
	X =  470.179  mm,	Y =   -318.103  mm,	Z =   -236.231  mm,
	W =  90.000 deg,	P =   0.000 deg,	R =   90.000 deg
};
P[3130]{
   GP1:
	UF : 0, UT : 6,		CONFIG : 'N U T, 0, 0, 0',
	X =  468.547  mm,	Y =   -315.184  mm,	Z =   -236.104  mm,
	W =  90.000 deg,	P =   0.000 deg,	R =   90.000 deg
};
P[3131]{
   GP1:
	UF : 0, UT : 6,		CONFIG : 'N U T, 0, 0, 0',
	X =  467.442  mm,	Y =   -313.499  mm,	Z =   -236.421  mm,
	W =  90.000 deg,	P =   0.000 deg,	R =   90.000 deg
};
P[3132]{
   GP1:
	UF : 0, UT : 6,		CONFIG : 'N U T, 0, 0, 0',
	X =  466.902  mm,	Y =   -312.524  mm,	Z =   -236.366  mm,
	W =  90.000 deg,	P =   0.000 deg,	R =   90.000 deg
};
P[3133]{
   GP1:
	UF : 0, UT : 6,		CONFIG : 'N U T, 0, 0, 0',
	X =  465.724  mm,	Y =   -310.259  mm,	Z =   -236.051  mm,
	W =  90.000 deg,	P =   0.000 deg,	R =   90.000 deg
};
P[3134]{
   GP1:
	UF : 0, UT : 6,		CONFIG : 'N U T, 0, 0, 0',
	X =  462.455  mm,	Y =   -304.923  mm,	Z =   -236.509  mm,
	W =  90.000 deg,	P =   0.000 deg,	R =   90.000 deg
};
P[3135]{
   GP1:
	UF : 0, UT : 6,		CONFIG : 'N U T, 0, 0, 0',
	X =  461.117  mm,	Y =   -302.322  mm,	Z =   -236.112  mm,
	W =  90.000 deg,	P =   0.000 deg,	R =   90.000 deg
};
P[3136]{
   GP1:
	UF : 0, UT : 6,		CONFIG : 'N U T, 0, 0, 0',
	X =  459.550  mm,	Y =   -299.871  mm,	Z =   -236.479  mm,
	W =  90.000 deg,	P =   0.000 deg,	R =   90.000 deg
};
P[3137]{
   GP1:
	UF : 0, UT : 6,		CONFIG : 'N U T, 0, 0, 0',
	X =  458.498  mm,	Y =   -297.980  mm,	Z =   -236.382  mm,
	W =  90.000 deg,	P =   0.000 deg,	R =   90.000 deg
};
P[3138]{
   GP1:
	UF : 0, UT : 6,		CONFIG : 'N U T, 0, 0, 0',
	X =  457.872  mm,	Y =   -296.943  mm,	Z =   -236.448  mm,
	W =  90.000 deg,	P =   0.000 deg,	R =   90.000 deg
};
P[3139]{
   GP1:
	UF : 0, UT : 6,		CONFIG : 'N U T, 0, 0, 0',
	X =  456.547  mm,	Y =   -294.555  mm,	Z =   -236.320  mm,
	W =  90.000 deg,	P =   0.000 deg,	R =   90.000 deg
};
P[3140]{
   GP1:
	UF : 0, UT : 6,		CONFIG : 'N U T, 0, 0, 0',
	X =  454.677  mm,	Y =   -291.318  mm,	Z =   -236.320  mm,
	W =  90.000 deg,	P =   0.000 deg,	R =   90.000 deg
};
P[3141]{
   GP1:
	UF : 0, UT : 6,		CONFIG : 'N U T, 0, 0, 0',
	X =  454.234  mm,	Y =   -290.583  mm,	Z =   -236.368  mm,
	W =  90.000 deg,	P =   0.000 deg,	R =   90.000 deg
};
P[3142]{
   GP1:
	UF : 0, UT : 6,		CONFIG : 'N U T, 0, 0, 0',
	X =  452.237  mm,	Y =   -287.074  mm,	Z =   -236.297  mm,
	W =  90.000 deg,	P =   0.000 deg,	R =   90.000 deg
};
P[3143]{
   GP1:
	UF : 0, UT : 6,		CONFIG : 'N U T, 0, 0, 0',
	X =  451.350  mm,	Y =   -285.562  mm,	Z =   -236.328  mm,
	W =  90.000 deg,	P =   0.000 deg,	R =   90.000 deg
};
P[3144]{
   GP1:
	UF : 0, UT : 6,		CONFIG : 'N U T, 0, 0, 0',
	X =  449.706  mm,	Y =   -282.695  mm,	Z =   -236.301  mm,
	W =  90.000 deg,	P =   0.000 deg,	R =   90.000 deg
};
P[3145]{
   GP1:
	UF : 0, UT : 6,		CONFIG : 'N U T, 0, 0, 0',
	X =  447.101  mm,	Y =   -278.322  mm,	Z =   -236.495  mm,
	W =  90.000 deg,	P =   0.000 deg,	R =   90.000 deg
};
P[3146]{
   GP1:
	UF : 0, UT : 6,		CONFIG : 'N U T, 0, 0, 0',
	X =  446.653  mm,	Y =   -277.554  mm,	Z =   -236.506  mm,
	W =  90.000 deg,	P =   0.000 deg,	R =   90.000 deg
};
P[3147]{
   GP1:
	UF : 0, UT : 6,		CONFIG : 'N U T, 0, 0, 0',
	X =  445.289  mm,	Y =   -275.164  mm,	Z =   -236.467  mm,
	W =  90.000 deg,	P =   0.000 deg,	R =   90.000 deg
};
P[3148]{
   GP1:
	UF : 0, UT : 6,		CONFIG : 'N U T, 0, 0, 0',
	X =  444.773  mm,	Y =   -274.241  mm,	Z =   -236.427  mm,
	W =  90.000 deg,	P =   0.000 deg,	R =   90.000 deg
};
P[3149]{
   GP1:
	UF : 0, UT : 6,		CONFIG : 'N U T, 0, 0, 0',
	X =  443.371  mm,	Y =   -271.687  mm,	Z =   -236.253  mm,
	W =  90.000 deg,	P =   0.000 deg,	R =   90.000 deg
};
P[3150]{
   GP1:
	UF : 0, UT : 6,		CONFIG : 'N U T, 0, 0, 0',
	X =  440.822  mm,	Y =   -267.250  mm,	Z =   -236.219  mm,
	W =  90.000 deg,	P =   0.000 deg,	R =   90.000 deg
};
P[3151]{
   GP1:
	UF : 0, UT : 6,		CONFIG : 'N U T, 0, 0, 0',
	X =  439.549  mm,	Y =   -265.240  mm,	Z =   -236.494  mm,
	W =  90.000 deg,	P =   0.000 deg,	R =   90.000 deg
};
P[3152]{
   GP1:
	UF : 0, UT : 6,		CONFIG : 'N U T, 0, 0, 0',
	X =  437.253  mm,	Y =   -261.131  mm,	Z =   -236.308  mm,
	W =  90.000 deg,	P =   0.000 deg,	R =   90.000 deg
};
P[3153]{
   GP1:
	UF : 0, UT : 6,		CONFIG : 'N U T, 0, 0, 0',
	X =  436.047  mm,	Y =   -258.958  mm,	Z =   -236.188  mm,
	W =  90.000 deg,	P =   0.000 deg,	R =   90.000 deg
};
P[3154]{
   GP1:
	UF : 0, UT : 6,		CONFIG : 'N U T, 0, 0, 0',
	X =  435.366  mm,	Y =   -257.755  mm,	Z =   -236.157  mm,
	W =  90.000 deg,	P =   0.000 deg,	R =   90.000 deg
};
P[3155]{
   GP1:
	UF : 0, UT : 6,		CONFIG : 'N U T, 0, 0, 0',
	X =  434.391  mm,	Y =   -256.258  mm,	Z =   -236.425  mm,
	W =  90.000 deg,	P =   0.000 deg,	R =   90.000 deg
};
P[3156]{
   GP1:
	UF : 0, UT : 6,		CONFIG : 'N U T, 0, 0, 0',
	X =  433.785  mm,	Y =   -255.204  mm,	Z =   -236.417  mm,
	W =  90.000 deg,	P =   0.000 deg,	R =   90.000 deg
};
P[3157]{
   GP1:
	UF : 0, UT : 6,		CONFIG : 'N U T, 0, 0, 0',
	X =  432.682  mm,	Y =   -253.326  mm,	Z =   -236.462  mm,
	W =  90.000 deg,	P =   0.000 deg,	R =   90.000 deg
};
P[3158]{
   GP1:
	UF : 0, UT : 6,		CONFIG : 'N U T, 0, 0, 0',
	X =  432.135  mm,	Y =   -252.408  mm,	Z =   -236.505  mm,
	W =  90.000 deg,	P =   0.000 deg,	R =   90.000 deg
};
P[3159]{
   GP1:
	UF : 0, UT : 6,		CONFIG : 'N U T, 0, 0, 0',
	X =  430.337  mm,	Y =   -249.170  mm,	Z =   -236.332  mm,
	W =  90.000 deg,	P =   0.000 deg,	R =   90.000 deg
};
P[3160]{
   GP1:
	UF : 0, UT : 6,		CONFIG : 'N U T, 0, 0, 0',
	X =  429.769  mm,	Y =   -248.131  mm,	Z =   -236.254  mm,
	W =  90.000 deg,	P =   0.000 deg,	R =   90.000 deg
};
P[3161]{
   GP1:
	UF : 0, UT : 6,		CONFIG : 'N U T, 0, 0, 0',
	X =  429.348  mm,	Y =   -247.471  mm,	Z =   -236.352  mm,
	W =  90.000 deg,	P =   0.000 deg,	R =   90.000 deg
};
P[3162]{
   GP1:
	UF : 0, UT : 6,		CONFIG : 'N U T, 0, 0, 0',
	X =  428.890  mm,	Y =   -246.615  mm,	Z =   -236.264  mm,
	W =  90.000 deg,	P =   0.000 deg,	R =   90.000 deg
};
P[3163]{
   GP1:
	UF : 0, UT : 6,		CONFIG : 'N U T, 0, 0, 0',
	X =  426.636  mm,	Y =   -242.550  mm,	Z =   -236.037  mm,
	W =  90.000 deg,	P =   0.000 deg,	R =   90.000 deg
};
P[3164]{
   GP1:
	UF : 0, UT : 6,		CONFIG : 'N U T, 0, 0, 0',
	X =  426.038  mm,	Y =   -241.779  mm,	Z =   -236.408  mm,
	W =  90.000 deg,	P =   0.000 deg,	R =   90.000 deg
};
P[3165]{
   GP1:
	UF : 0, UT : 6,		CONFIG : 'N U T, 0, 0, 0',
	X =  425.607  mm,	Y =   -240.797  mm,	Z =   -236.076  mm,
	W =  90.000 deg,	P =   0.000 deg,	R =   90.000 deg
};
P[3166]{
   GP1:
	UF : 0, UT : 6,		CONFIG : 'N U T, 0, 0, 0',
	X =  424.035  mm,	Y =   -238.243  mm,	Z =   -236.313  mm,
	W =  90.000 deg,	P =   0.000 deg,	R =   90.000 deg
};
P[3167]{
   GP1:
	UF : 0, UT : 6,		CONFIG : 'N U T, 0, 0, 0',
	X =  423.311  mm,	Y =   -237.117  mm,	Z =   -236.494  mm,
	W =  90.000 deg,	P =   0.000 deg,	R =   90.000 deg
};
P[3168]{
   GP1:
	UF : 0, UT : 6,		CONFIG : 'N U T, 0, 0, 0',
	X =  422.742  mm,	Y =   -236.079  mm,	Z =   -236.420  mm,
	W =  90.000 deg,	P =   0.000 deg,	R =   90.000 deg
};
P[3169]{
   GP1:
	UF : 0, UT : 6,		CONFIG : 'N U T, 0, 0, 0',
	X =  422.185  mm,	Y =   -235.164  mm,	Z =   -236.487  mm,
	W =  90.000 deg,	P =   0.000 deg,	R =   90.000 deg
};
P[3170]{
   GP1:
	UF : 0, UT : 6,		CONFIG : 'N U T, 0, 0, 0',
	X =  421.846  mm,	Y =   -234.239  mm,	Z =   -236.017  mm,
	W =  90.000 deg,	P =   0.000 deg,	R =   90.000 deg
};
P[3171]{
   GP1:
	UF : 0, UT : 6,		CONFIG : 'N U T, 0, 0, 0',
	X =  421.354  mm,	Y =   -233.685  mm,	Z =   -236.432  mm,
	W =  90.000 deg,	P =   0.000 deg,	R =   90.000 deg
};
P[3172]{
   GP1:
	UF : 0, UT : 6,		CONFIG : 'N U T, 0, 0, 0',
	X =  420.263  mm,	Y =   -231.706  mm,	Z =   -236.309  mm,
	W =  90.000 deg,	P =   0.000 deg,	R =   90.000 deg
};
P[3173]{
   GP1:
	UF : 0, UT : 6,		CONFIG : 'N U T, 0, 0, 0',
	X =  419.547  mm,	Y =   -230.374  mm,	Z =   -236.177  mm,
	W =  90.000 deg,	P =   0.000 deg,	R =   90.000 deg
};
P[3174]{
   GP1:
	UF : 0, UT : 6,		CONFIG : 'N U T, 0, 0, 0',
	X =  418.540  mm,	Y =   -228.547  mm,	Z =   -236.062  mm,
	W =  90.000 deg,	P =   0.000 deg,	R =   90.000 deg
};
P[3175]{
   GP1:
	UF : 0, UT : 6,		CONFIG : 'N U T, 0, 0, 0',
	X =  417.729  mm,	Y =   -227.381  mm,	Z =   -236.397  mm,
	W =  90.000 deg,	P =   0.000 deg,	R =   90.000 deg
};
P[3176]{
   GP1:
	UF : 0, UT : 6,		CONFIG : 'N U T, 0, 0, 0',
	X =  417.237  mm,	Y =   -226.307  mm,	Z =   -236.087  mm,
	W =  90.000 deg,	P =   0.000 deg,	R =   90.000 deg
};
P[3177]{
   GP1:
	UF : 0, UT : 6,		CONFIG : 'N U T, 0, 0, 0',
	X =  416.602  mm,	Y =   -225.198  mm,	Z =   -236.074  mm,
	W =  90.000 deg,	P =   0.000 deg,	R =   90.000 deg
};
P[3178]{
   GP1:
	UF : 0, UT : 6,		CONFIG : 'N U T, 0, 0, 0',
	X =  416.038  mm,	Y =   -224.516  mm,	Z =   -236.487  mm,
	W =  90.000 deg,	P =   0.000 deg,	R =   90.000 deg
};
P[3179]{
   GP1:
	UF : 0, UT : 6,		CONFIG : 'N U T, 0, 0, 0',
	X =  413.995  mm,	Y =   -220.945  mm,	Z =   -236.440  mm,
	W =  90.000 deg,	P =   0.000 deg,	R =   90.000 deg
};
P[3180]{
   GP1:
	UF : 0, UT : 6,		CONFIG : 'N U T, 0, 0, 0',
	X =  413.625  mm,	Y =   -220.345  mm,	Z =   -236.498  mm,
	W =  90.000 deg,	P =   0.000 deg,	R =   90.000 deg
};
P[3181]{
   GP1:
	UF : 0, UT : 6,		CONFIG : 'N U T, 0, 0, 0',
	X =  411.729  mm,	Y =   -216.911  mm,	Z =   -236.287  mm,
	W =  90.000 deg,	P =   0.000 deg,	R =   90.000 deg
};
P[3182]{
   GP1:
	UF : 0, UT : 6,		CONFIG : 'N U T, 0, 0, 0',
	X =  411.113  mm,	Y =   -215.668  mm,	Z =   -236.041  mm,
	W =  90.000 deg,	P =   0.000 deg,	R =   90.000 deg
};
P[3183]{
   GP1:
	UF : 0, UT : 6,		CONFIG : 'N U T, 0, 0, 0',
	X =  410.660  mm,	Y =   -214.893  mm,	Z =   -236.055  mm,
	W =  90.000 deg,	P =   0.000 deg,	R =   90.000 deg
};
P[3184]{
   GP1:
	UF : 0, UT : 6,		CONFIG : 'N U T, 0, 0, 0',
	X =  410.172  mm,	Y =   -214.352  mm,	Z =   -236.479  mm,
	W =  90.000 deg,	P =   0.000 deg,	R =   90.000 deg
};
P[3185]{
   GP1:
	UF : 0, UT : 6,		CONFIG : 'N U T, 0, 0, 0',
	X =  409.070  mm,	Y =   -212.287  mm,	Z =   -236.260  mm,
	W =  90.000 deg,	P =   0.000 deg,	R =   90.000 deg
};
P[3186]{
   GP1:
	UF : 0, UT : 6,		CONFIG : 'N U T, 0, 0, 0',
	X =  405.949  mm,	Y =   -207.005  mm,	Z =   -236.432  mm,
	W =  90.000 deg,	P =   0.000 deg,	R =   90.000 deg
};
P[3187]{
   GP1:
	UF : 0, UT : 6,		CONFIG : 'N U T, 0, 0, 0',
	X =  403.776  mm,	Y =   -203.175  mm,	Z =   -236.339  mm,
	W =  90.000 deg,	P =   0.000 deg,	R =   90.000 deg
};
P[3188]{
   GP1:
	UF : 0, UT : 6,		CONFIG : 'N U T, 0, 0, 0',
	X =  402.283  mm,	Y =   -200.497  mm,	Z =   -236.211  mm,
	W =  90.000 deg,	P =   0.000 deg,	R =   90.000 deg
};
P[3189]{
   GP1:
	UF : 0, UT : 6,		CONFIG : 'N U T, 0, 0, 0',
	X =  401.755  mm,	Y =   -199.688  mm,	Z =   -236.359  mm,
	W =  90.000 deg,	P =   0.000 deg,	R =   90.000 deg
};
P[3190]{
   GP1:
	UF : 0, UT : 6,		CONFIG : 'N U T, 0, 0, 0',
	X =  401.172  mm,	Y =   -198.643  mm,	Z =   -236.311  mm,
	W =  90.000 deg,	P =   0.000 deg,	R =   90.000 deg
};
P[3191]{
   GP1:
	UF : 0, UT : 6,		CONFIG : 'N U T, 0, 0, 0',
	X =  400.173  mm,	Y =   -196.923  mm,	Z =   -236.324  mm,
	W =  90.000 deg,	P =   0.000 deg,	R =   90.000 deg
};
P[3192]{
   GP1:
	UF : 0, UT : 6,		CONFIG : 'N U T, 0, 0, 0',
	X =  399.182  mm,	Y =   -195.254  mm,	Z =   -236.388  mm,
	W =  90.000 deg,	P =   0.000 deg,	R =   90.000 deg
};
P[3193]{
   GP1:
	UF : 0, UT : 6,		CONFIG : 'N U T, 0, 0, 0',
	X =  398.400  mm,	Y =   -193.951  mm,	Z =   -236.462  mm,
	W =  90.000 deg,	P =   0.000 deg,	R =   90.000 deg
};
P[3194]{
   GP1:
	UF : 0, UT : 6,		CONFIG : 'N U T, 0, 0, 0',
	X =  397.319  mm,	Y =   -192.048  mm,	Z =   -236.420  mm,
	W =  90.000 deg,	P =   0.000 deg,	R =   90.000 deg
};
P[3195]{
   GP1:
	UF : 0, UT : 6,		CONFIG : 'N U T, 0, 0, 0',
	X =  396.424  mm,	Y =   -190.499  mm,	Z =   -236.421  mm,
	W =  90.000 deg,	P =   0.000 deg,	R =   90.000 deg
};
P[3196]{
   GP1:
	UF : 0, UT : 6,		CONFIG : 'N U T, 0, 0, 0',
	X =  395.868  mm,	Y =   -189.559  mm,	Z =   -236.452  mm,
	W =  90.000 deg,	P =   0.000 deg,	R =   90.000 deg
};
P[3197]{
   GP1:
	UF : 0, UT : 6,		CONFIG : 'N U T, 0, 0, 0',
	X =  394.876  mm,	Y =   -187.860  mm,	Z =   -236.479  mm,
	W =  90.000 deg,	P =   0.000 deg,	R =   90.000 deg
};
P[3198]{
   GP1:
	UF : 0, UT : 6,		CONFIG : 'N U T, 0, 0, 0',
	X =  394.097  mm,	Y =   -186.491  mm,	Z =   -236.452  mm,
	W =  90.000 deg,	P =   0.000 deg,	R =   90.000 deg
};
P[3199]{
   GP1:
	UF : 0, UT : 6,		CONFIG : 'N U T, 0, 0, 0',
	X =  393.502  mm,	Y =   -185.416  mm,	Z =   -236.390  mm,
	W =  90.000 deg,	P =   0.000 deg,	R =   90.000 deg
};
P[3200]{
   GP1:
	UF : 0, UT : 6,		CONFIG : 'N U T, 0, 0, 0',
	X =  392.903  mm,	Y =   -184.170  mm,	Z =   -236.098  mm,
	W =  90.000 deg,	P =   0.000 deg,	R =   90.000 deg
};
P[3201]{
   GP1:
	UF : 0, UT : 6,		CONFIG : 'N U T, 0, 0, 0',
	X =  391.649  mm,	Y =   -182.107  mm,	Z =   -236.249  mm,
	W =  90.000 deg,	P =   0.000 deg,	R =   90.000 deg
};
P[3202]{
   GP1:
	UF : 0, UT : 6,		CONFIG : 'N U T, 0, 0, 0',
	X =  390.355  mm,	Y =   -180.021  mm,	Z =   -236.466  mm,
	W =  90.000 deg,	P =   0.000 deg,	R =   90.000 deg
};
P[3203]{
   GP1:
	UF : 0, UT : 6,		CONFIG : 'N U T, 0, 0, 0',
	X =  387.951  mm,	Y =   -175.769  mm,	Z =   -236.341  mm,
	W =  90.000 deg,	P =   0.000 deg,	R =   90.000 deg
};
P[3204]{
   GP1:
	UF : 0, UT : 6,		CONFIG : 'N U T, 0, 0, 0',
	X =  385.398  mm,	Y =   -171.250  mm,	Z =   -236.206  mm,
	W =  90.000 deg,	P =   0.000 deg,	R =   90.000 deg
};
P[3205]{
   GP1:
	UF : 0, UT : 6,		CONFIG : 'N U T, 0, 0, 0',
	X =  383.021  mm,	Y =   -167.308  mm,	Z =   -236.452  mm,
	W =  90.000 deg,	P =   0.000 deg,	R =   90.000 deg
};
P[3206]{
   GP1:
	UF : 0, UT : 6,		CONFIG : 'N U T, 0, 0, 0',
	X =  381.764  mm,	Y =   -165.174  mm,	Z =   -236.511  mm,
	W =  90.000 deg,	P =   0.000 deg,	R =   90.000 deg
};
P[3207]{
   GP1:
	UF : 0, UT : 6,		CONFIG : 'N U T, 0, 0, 0',
	X =  380.817  mm,	Y =   -163.283  mm,	Z =   -236.162  mm,
	W =  90.000 deg,	P =   0.000 deg,	R =   90.000 deg
};
P[3208]{
   GP1:
	UF : 0, UT : 6,		CONFIG : 'N U T, 0, 0, 0',
	X =  380.351  mm,	Y =   -162.620  mm,	Z =   -236.361  mm,
	W =  90.000 deg,	P =   0.000 deg,	R =   90.000 deg
};
P[3209]{
   GP1:
	UF : 0, UT : 6,		CONFIG : 'N U T, 0, 0, 0',
	X =  379.247  mm,	Y =   -160.676  mm,	Z =   -236.316  mm,
	W =  90.000 deg,	P =   0.000 deg,	R =   90.000 deg
};
P[3210]{
   GP1:
	UF : 0, UT : 6,		CONFIG : 'N U T, 0, 0, 0',
	X =  378.744  mm,	Y =   -159.629  mm,	Z =   -236.071  mm,
	W =  90.000 deg,	P =   0.000 deg,	R =   90.000 deg
};
P[3211]{
   GP1:
	UF : 0, UT : 6,		CONFIG : 'N U T, 0, 0, 0',
	X =  376.743  mm,	Y =   -156.129  mm,	Z =   -236.020  mm,
	W =  90.000 deg,	P =   0.000 deg,	R =   90.000 deg
};
P[3212]{
   GP1:
	UF : 0, UT : 6,		CONFIG : 'N U T, 0, 0, 0',
	X =  375.969  mm,	Y =   -155.020  mm,	Z =   -236.347  mm,
	W =  90.000 deg,	P =   0.000 deg,	R =   90.000 deg
};
P[3213]{
   GP1:
	UF : 0, UT : 6,		CONFIG : 'N U T, 0, 0, 0',
	X =  375.333  mm,	Y =   -153.875  mm,	Z =   -236.286  mm,
	W =  90.000 deg,	P =   0.000 deg,	R =   90.000 deg
};
P[3214]{
   GP1:
	UF : 0, UT : 6,		CONFIG : 'N U T, 0, 0, 0',
	X =  374.357  mm,	Y =   -152.153  mm,	Z =   -236.242  mm,
	W =  90.000 deg,	P =   0.000 deg,	R =   90.000 deg
};
P[3215]{
   GP1:
	UF : 0, UT : 6,		CONFIG : 'N U T, 0, 0, 0',
	X =  372.698  mm,	Y =   -149.350  mm,	Z =   -236.339  mm,
	W =  90.000 deg,	P =   0.000 deg,	R =   90.000 deg
};
P[3216]{
   GP1:
	UF : 0, UT : 6,		CONFIG : 'N U T, 0, 0, 0',
	X =  368.549  mm,	Y =   -142.281  mm,	Z =   -236.503  mm,
	W =  90.000 deg,	P =   0.000 deg,	R =   90.000 deg
};
P[3217]{
   GP1:
	UF : 0, UT : 6,		CONFIG : 'N U T, 0, 0, 0',
	X =  367.899  mm,	Y =   -141.052  mm,	Z =   -236.359  mm,
	W =  90.000 deg,	P =   0.000 deg,	R =   90.000 deg
};
P[3218]{
   GP1:
	UF : 0, UT : 6,		CONFIG : 'N U T, 0, 0, 0',
	X =  367.592  mm,	Y =   -140.381  mm,	Z =   -236.163  mm,
	W =  90.000 deg,	P =   0.000 deg,	R =   90.000 deg
};
P[3219]{
   GP1:
	UF : 0, UT : 6,		CONFIG : 'N U T, 0, 0, 0',
	X =  366.850  mm,	Y =   -139.318  mm,	Z =   -236.475  mm,
	W =  90.000 deg,	P =   0.000 deg,	R =   90.000 deg
};
P[3220]{
   GP1:
	UF : 0, UT : 6,		CONFIG : 'N U T, 0, 0, 0',
	X =  365.974  mm,	Y =   -137.729  mm,	Z =   -236.376  mm,
	W =  90.000 deg,	P =   0.000 deg,	R =   90.000 deg
};
P[3221]{
   GP1:
	UF : 0, UT : 6,		CONFIG : 'N U T, 0, 0, 0',
	X =  363.425  mm,	Y =   -133.317  mm,	Z =   -236.380  mm,
	W =  90.000 deg,	P =   0.000 deg,	R =   90.000 deg
};
P[3222]{
   GP1:
	UF : 0, UT : 6,		CONFIG : 'N U T, 0, 0, 0',
	X =  362.686  mm,	Y =   -131.801  mm,	Z =   -236.048  mm,
	W =  90.000 deg,	P =   0.000 deg,	R =   90.000 deg
};
P[3223]{
   GP1:
	UF : 0, UT : 6,		CONFIG : 'N U T, 0, 0, 0',
	X =  361.274  mm,	Y =   -129.357  mm,	Z =   -236.049  mm,
	W =  90.000 deg,	P =   0.000 deg,	R =   90.000 deg
};
P[3224]{
   GP1:
	UF : 0, UT : 6,		CONFIG : 'N U T, 0, 0, 0',
	X =  360.867  mm,	Y =   -128.750  mm,	Z =   -236.185  mm,
	W =  90.000 deg,	P =   0.000 deg,	R =   90.000 deg
};
P[3225]{
   GP1:
	UF : 0, UT : 6,		CONFIG : 'N U T, 0, 0, 0',
	X =  359.775  mm,	Y =   -126.789  mm,	Z =   -236.086  mm,
	W =  90.000 deg,	P =   0.000 deg,	R =   90.000 deg
};
P[3226]{
   GP1:
	UF : 0, UT : 6,		CONFIG : 'N U T, 0, 0, 0',
	X =  358.196  mm,	Y =   -124.234  mm,	Z =   -236.341  mm,
	W =  90.000 deg,	P =   0.000 deg,	R =   90.000 deg
};
P[3227]{
   GP1:
	UF : 0, UT : 6,		CONFIG : 'N U T, 0, 0, 0',
	X =  357.493  mm,	Y =   -122.993  mm,	Z =   -236.306  mm,
	W =  90.000 deg,	P =   0.000 deg,	R =   90.000 deg
};
P[3228]{
   GP1:
	UF : 0, UT : 6,		CONFIG : 'N U T, 0, 0, 0',
	X =  356.675  mm,	Y =   -121.501  mm,	Z =   -236.203  mm,
	W =  90.000 deg,	P =   0.000 deg,	R =   90.000 deg
};
P[3229]{
   GP1:
	UF : 0, UT : 6,		CONFIG : 'N U T, 0, 0, 0',
	X =  354.180  mm,	Y =   -117.458  mm,	Z =   -236.282  mm,
	W =  90.000 deg,	P =   0.000 deg,	R =   90.000 deg
};
P[3230]{
   GP1:
	UF : 0, UT : 6,		CONFIG : 'N U T, 0, 0, 0',
	X =  353.504  mm,	Y =   -116.554  mm,	Z =   -236.351  mm,
	W =  90.000 deg,	P =   0.000 deg,	R =   90.000 deg
};
P[3231]{
   GP1:
	UF : 0, UT : 6,		CONFIG : 'N U T, 0, 0, 0',
	X =  352.989  mm,	Y =   -115.735  mm,	Z =   -236.027  mm,
	W =  90.000 deg,	P =   0.000 deg,	R =   90.000 deg
};
P[3232]{
   GP1:
	UF : 0, UT : 6,		CONFIG : 'N U T, 0, 0, 0',
	X =  352.209  mm,	Y =   -115.216  mm,	Z =   -236.403  mm,
	W =  90.000 deg,	P =   0.000 deg,	R =   90.000 deg
};
P[3233]{
   GP1:
	UF : 0, UT : 6,		CONFIG : 'N U T, 0, 0, 0',
